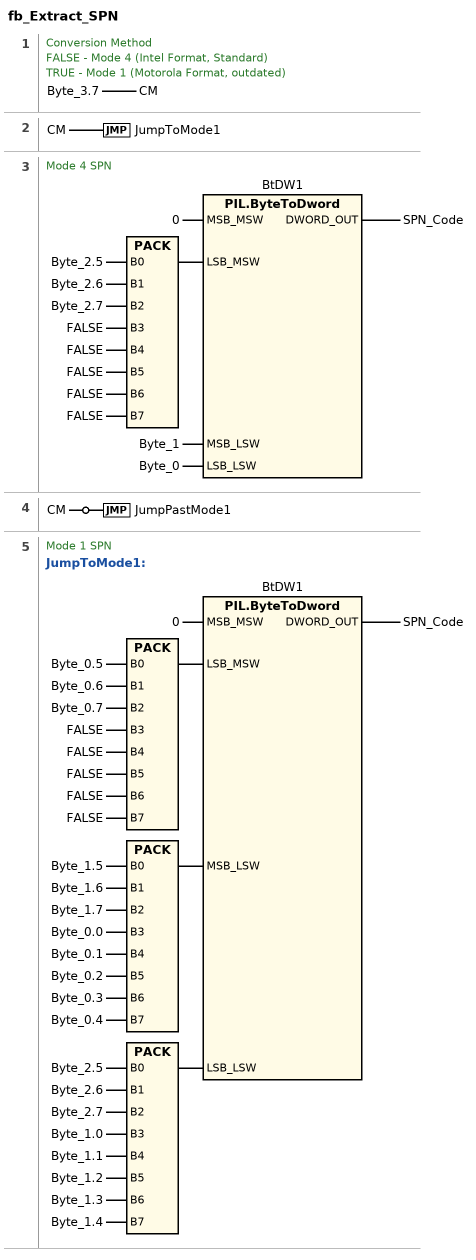
// NETWORK 1
// 					Conversion Method
// FALSE - Mode 4 (Intel Format, Standard)
// TRUE - Mode 1 (Motorola Format, outdated)
//
CM := Byte_3.7;

// NETWORK 2
IF CM THEN JMP JumpToMode1; END_IF

// NETWORK 3
// Mode 4 SPN
BtDW1(
    MSB_MSW := 0,
    LSB_MSW := PACK(B0 := Byte_2.5, B1 := Byte_2.6, B2 := Byte_2.7, B3 := FALSE, B4 := FALSE, B5 := FALSE, B6 := FALSE, B7 := FALSE),
    MSB_LSW := Byte_1,
    LSB_LSW := Byte_0); // PIL.ByteToDword
SPN_Code := BtDW1.DWORD_OUT;

// NETWORK 4
IF NOT CM THEN JMP JumpPastMode1; END_IF

// NETWORK 5
// Mode 1 SPN
JumpToMode1:
BtDW1(
    MSB_MSW := 0,
    LSB_MSW := PACK(B0 := Byte_0.5, B1 := Byte_0.6, B2 := Byte_0.7, B3 := FALSE, B4 := FALSE, B5 := FALSE, B6 := FALSE, B7 := FALSE),
    MSB_LSW := PACK(B0 := Byte_1.5, B1 := Byte_1.6, B2 := Byte_1.7, B3 := Byte_0.0, B4 := Byte_0.1, B5 := Byte_0.2, B6 := Byte_0.3, B7 := Byte_0.4),
    LSB_LSW := PACK(B0 := Byte_2.5, B1 := Byte_2.6, B2 := Byte_2.7, B3 := Byte_1.0, B4 := Byte_1.1, B5 := Byte_1.2, B6 := Byte_1.3, B7 := Byte_1.4)); // PIL.ByteToDword
SPN_Code := BtDW1.DWORD_OUT;

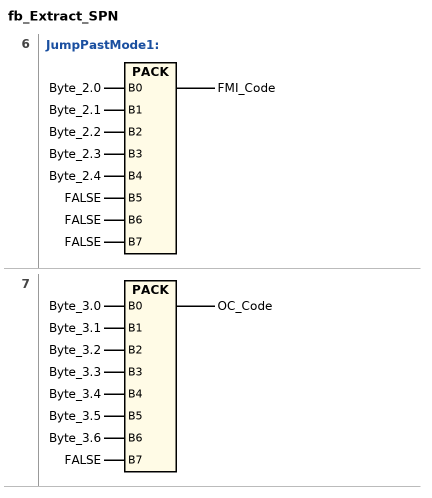
// NETWORK 6
JumpPastMode1:
FMI_Code := PACK(B0 := Byte_2.0, B1 := Byte_2.1, B2 := Byte_2.2, B3 := Byte_2.3, B4 := Byte_2.4, B5 := FALSE, B6 := FALSE, B7 := FALSE);

// NETWORK 7
OC_Code := PACK(B0 := Byte_3.0, B1 := Byte_3.1, B2 := Byte_3.2, B3 := Byte_3.3, B4 := Byte_3.4, B5 := Byte_3.5, B6 := Byte_3.6, B7 := FALSE);

END_FUNCTION_BLOCK

// Device/Application/App_PLC/CAN Comms/Engine Comms/Pack2bits
FUNCTION_BLOCK Pack2bits
VAR_INPUT
	LS_bit: BOOL;
	MS_bit: BOOL;
END_VAR
VAR_OUTPUT
	Out: BYTE;
END_VAR
VAR
END_VAR

IF LS_bit=TRUE THEN Out:=1; ELSE Out:=0; END_IF
IF MS_bit=TRUE THEN Out:=Out+2; ELSE Out:=Out; END_IF

END_FUNCTION_BLOCK

// Device/Application/App_PLC/CAN Comms/Engine Comms/PLC_DM1_Condition
FUNCTION_BLOCK PLC_DM1_Condition

(*Function block to look for an active SPN that is contained within the Error codes array [1..15]
The ConditionActive ouptut is used when you want to identify a SPN with a certain FMI
The SPNActive output is TRUE when the requested SPN is contained anywhere withing the array*)

VAR_INPUT
	ActiveErrCount: BYTE;
	ReqSPN: DWORD;
	ReqFMI: BYTE;
END_VAR
VAR_OUTPUT
	SPNActive: BOOL;
	ConditionAcitve: BOOL;
END_VAR
VAR
(*Temporary Variables*)
	SPNActive_1: BOOL;
	SPNActive_2: BOOL;
	SPNActive_3: BOOL;
	SPNActive_4: BOOL;
	SPNActive_5: BOOL;
	SPNActive_6: BOOL;
	SPNActive_7: BOOL;	(*  *)
	SPNActive_8: BOOL;	(*  *)
END_VAR
VAR // added by the converter: edge detectors and wires of the graphical bodies
    _w1, _w2, _w3, _w4, _w5, _w6, _w7, _w8 : BOOL;
END_VAR

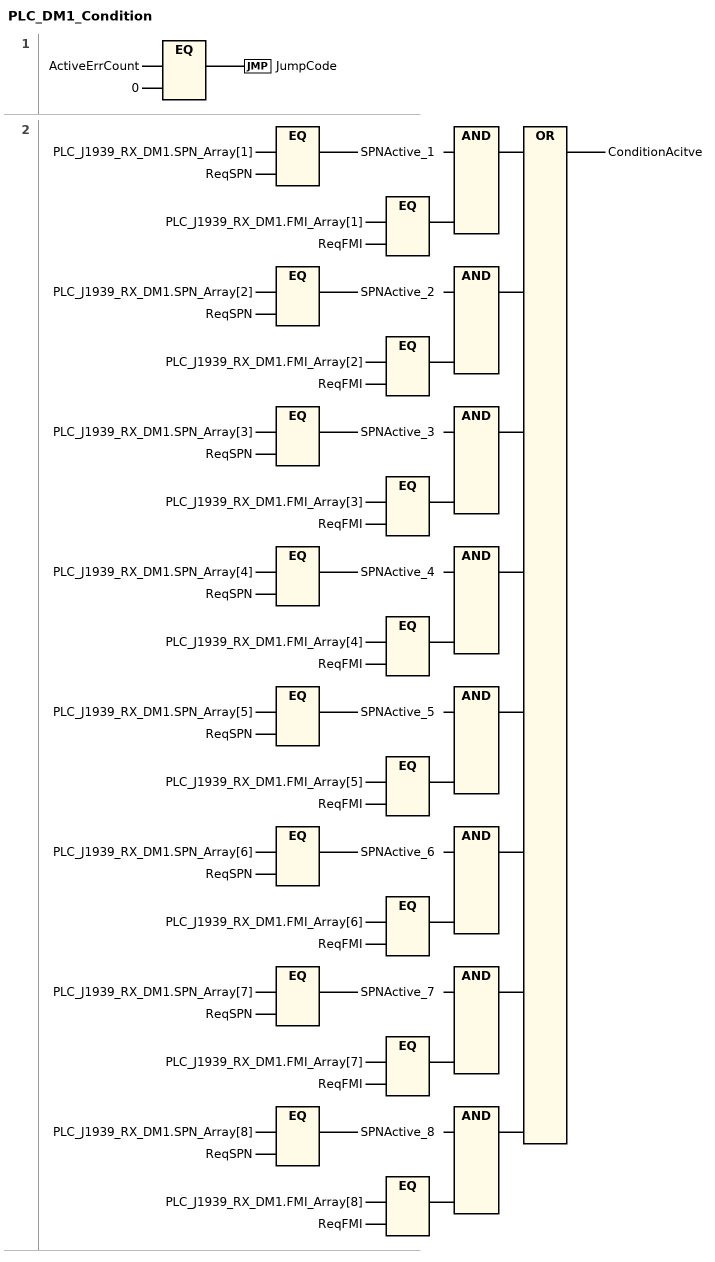
// NETWORK 1
IF ActiveErrCount = 0 THEN JMP JumpCode; END_IF

// NETWORK 2
_w1 := PLC_J1939_RX_DM1.SPN_Array[1] = ReqSPN;
SPNActive_1 := _w1;
_w2 := PLC_J1939_RX_DM1.SPN_Array[2] = ReqSPN;
SPNActive_2 := _w2;
_w3 := PLC_J1939_RX_DM1.SPN_Array[3] = ReqSPN;
SPNActive_3 := _w3;
_w4 := PLC_J1939_RX_DM1.SPN_Array[4] = ReqSPN;
SPNActive_4 := _w4;
_w5 := PLC_J1939_RX_DM1.SPN_Array[5] = ReqSPN;
SPNActive_5 := _w5;
_w6 := PLC_J1939_RX_DM1.SPN_Array[6] = ReqSPN;
SPNActive_6 := _w6;
_w7 := PLC_J1939_RX_DM1.SPN_Array[7] = ReqSPN;
SPNActive_7 := _w7;
_w8 := PLC_J1939_RX_DM1.SPN_Array[8] = ReqSPN;
SPNActive_8 := _w8;
ConditionAcitve := _w1 AND PLC_J1939_RX_DM1.FMI_Array[1] = ReqFMI OR _w2 AND PLC_J1939_RX_DM1.FMI_Array[2] = ReqFMI OR _w3 AND PLC_J1939_RX_DM1.FMI_Array[3] = ReqFMI OR _w4 AND PLC_J1939_RX_DM1.FMI_Array[4] = ReqFMI OR _w5 AND PLC_J1939_RX_DM1.FMI_Array[5] = ReqFMI OR _w6 AND PLC_J1939_RX_DM1.FMI_Array[6] = ReqFMI OR _w7 AND PLC_J1939_RX_DM1.FMI_Array[7] = ReqFMI OR _w8 AND PLC_J1939_RX_DM1.FMI_Array[8] = ReqFMI;

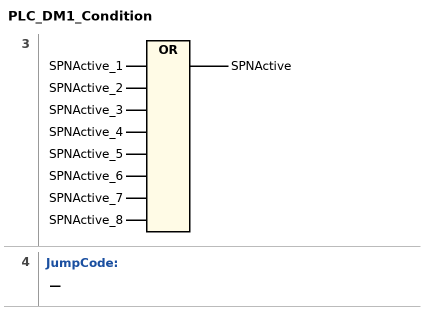
// NETWORK 3
SPNActive := SPNActive_1 OR SPNActive_2 OR SPNActive_3 OR SPNActive_4 OR SPNActive_5 OR SPNActive_6 OR SPNActive_7 OR SPNActive_8;

// NETWORK 4
JumpCode: ;

END_FUNCTION_BLOCK

// Device/Application/App_Common/Machine/APP_WARNINGS_ERRORS
PROGRAM APP_WARNINGS_ERRORS
VAR_INPUT
	TOTAL_ERRORS:INT;
	TOTAL_WARNINGS:INT;	
END_VAR
VAR
	HEADER_MSG_SWT_TON: TON;
	HEADER_MSG_SWT: WORD;
	HEADER_MSG_ENA: BOOL:=TRUE;

END_VAR
VAR_OUTPUT
	ERRORS_ACTIVE: BOOL;
	WARNINGS_ACTIVE: BOOL;
END_VAR


//TOTAL_ERRORS:=MAIN_ERRORS_COUNT+DIAG_IO_ERRORS_COUNT;

IF TOTAL_ERRORS > 0 THEN
	ERRORS_ACTIVE:=TRUE;
ELSE
	ERRORS_ACTIVE:=FALSE;
END_IF

IF TOTAL_WARNINGS > 0 THEN
	WARNINGS_ACTIVE:=TRUE;
ELSE
	WARNINGS_ACTIVE:=FALSE;
END_IF

IF HEADER_MSG_ENA THEN
	HEADER_MSG_SWT_TON(IN:=NOT(HEADER_MSG_SWT_TON.Q));
	
	IF HEADER_MSG_SWT_TON.Q THEN
		IF HEADER_MSG_SWT < 2 THEN
			HEADER_MSG_SWT:=HEADER_MSG_SWT+1;	
		ELSE
			HEADER_MSG_SWT:=0;		
		END_IF	
	END_IF

	IF GVL_Alarms.EMERGENCY_STOP_COMMON AND HEADER_MSG_SWT = 1 THEN
		NVL_Viz.Sections.Footer.Header_Message_Str:='ESTOP ACTIVE';
		NVL_Viz.Sections.Footer.Header_Message_Colour:=16#FFFF0000;
		NVL_Viz.Sections.Footer.Header_Message_Show:=TRUE;
		HEADER_MSG_SWT_TON.PT:=T#2000MS;
	ELSIF GVL_Alarms.ETHERNET_PLC_COMMON_FAILURE AND HEADER_MSG_SWT = 2 THEN
		NVL_Viz.Sections.Footer.Header_Message_Str:='PLCS OFFLINE';
		NVL_Viz.Sections.Footer.Header_Message_Colour:=16#FFFF0000;
		NVL_Viz.Sections.Footer.Header_Message_Show:=TRUE;
		HEADER_MSG_SWT_TON.PT:=T#3000MS;
	ELSE
		NVL_Viz.Sections.Footer.Header_Message_Str:='';
		NVL_Viz.Sections.Footer.Header_Message_Colour:=16#FF000000;
		NVL_Viz.Sections.Footer.Header_Message_Show:=FALSE;	
		HEADER_MSG_SWT_TON.PT:=T#1000MS;
	END_IF
ELSE
	NVL_Viz.Sections.Footer.Header_Message_Show:=FALSE;	
END_IF

END_PROGRAM

// Device/Application/App_Common/Machine/SIREN_BEACONS
PROGRAM SIREN_BEACONS
VAR_INPUT
	ESTOP_ACTIVE: BOOL;
	ERRORS_ACTIVE: BOOL;
	WARNINGS_ACTIVE: BOOL;
END_VAR
VAR
	SIREN_BLIP_PU_TON: TON;
	PRE_START_TON: TON;	
	
	SIREN_ALARMS: BOOL:=FALSE;
	SIREN_WARNINGS: BOOL:=FALSE;

	SIREN_PU_BLIP: BOOL;
	BEACON_PU_BLIP: BOOL;	
	
	BEACON_DEADMAN: BOOL;
	SIREN_DEADMAN: BOOL;
	SIREN_ESTOP: BOOL;
	TEST_SIREN: BOOL;
	TEST_BEACON: BOOL;
	
	SIREN_ALARMS_BLINK: DUTY_CYCLE;
	SIREN_WARNINGS_BLINK: DUTY_CYCLE;
END_VAR

VAR_OUTPUT
	SIREN_OUT: BOOL;
	BEACON_OUT: BOOL;
	PRESTART_TIMER_ACTIVE: BOOL;	
	PRESTART_TIMER_DONE: BOOL;
END_VAR
VAR // added by the converter: edge detectors and wires of the graphical bodies
    _w1 : BOOL;
END_VAR

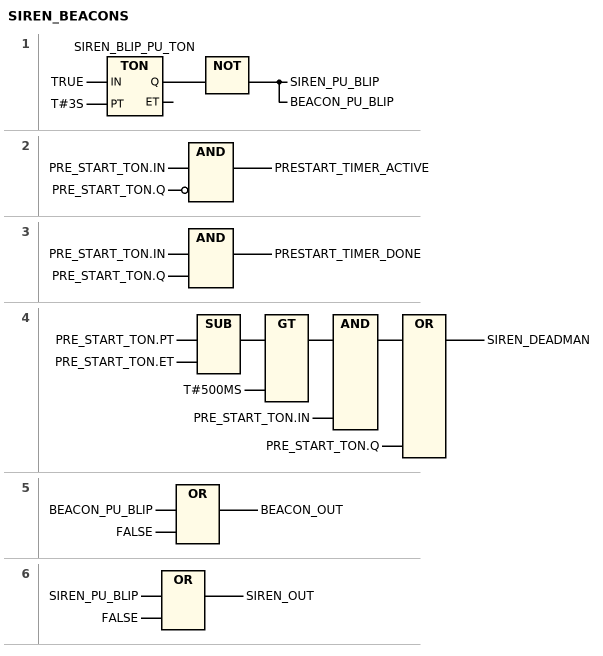
// NETWORK 1
SIREN_BLIP_PU_TON(IN := TRUE, PT := T#3S); // TON
_w1 := NOT SIREN_BLIP_PU_TON.Q;
SIREN_PU_BLIP := _w1;
BEACON_PU_BLIP := _w1;

// NETWORK 2
PRESTART_TIMER_ACTIVE := PRE_START_TON.IN AND NOT PRE_START_TON.Q;

// NETWORK 3
PRESTART_TIMER_DONE := PRE_START_TON.IN AND PRE_START_TON.Q;

// NETWORK 4
SIREN_DEADMAN := PRE_START_TON.PT - PRE_START_TON.ET > T#500MS AND PRE_START_TON.IN OR PRE_START_TON.Q;

// NETWORK 5
BEACON_OUT := BEACON_PU_BLIP OR FALSE;

// NETWORK 6
SIREN_OUT := SIREN_PU_BLIP OR FALSE;

END_PROGRAM

// Device/Application/App_Common/Nav/Page Control/AutoManSelButtons
PROGRAM AutoManSelButtons
VAR_INPUT
	Enable: BOOL;	
END_VAR

VAR
	Mimic_Halo_Sel_Max: WORD:=6;
	NavUpShow_TP: TP;
	NavDownShow_TP: TP;
	NavCircleShow_TP: TP;
	TailConv_RectIcon_FB: RectIcon;
	SideTransfer_RectIcon_FB: RectIcon;
	SideConveyor_RectIcon_FB: RectIcon;
	CollectConveyor_RectIcon_FB: RectIcon;
	Drum_RectIcon_FB: RectIcon;
	Feeder_RectIcon_FB: RectIcon;
	NavLeftShow_TP: TP;
	NavRightShow_TP: TP;
	AUTOSTOP_DUTY_CYCLE: DUTY_CYCLE;
	AUTOSTART_DUTY_CYCLE: DUTY_CYCLE;
	AutoActiveCommon: BOOL;
	
	PWM_Op_Status_FB_0: PWM_Op_Status_FB;
	PWM_Op_Status_FB_1: PWM_Op_Status_FB;
	PWM_Op_Status_FB_2: PWM_Op_Status_FB;
	PWM_Op_Status_FB_3: PWM_Op_Status_FB;
	PWM_Op_Status_FB_4: PWM_Op_Status_FB;
	PWM_Op_Status_FB_5: PWM_Op_Status_FB;	
	PWM_Op_Status_FB_: PWM_Op_Status_FB;
	
	PWM_Op_SideConveyor_Status_Str: STRING;
	PWM_Op_SideTransfer_Status_Str: STRING;	
	PWM_Op_TailConveyor_Status_Str: STRING;
	PWM_Op_CollectionConveyor_Status_Str: STRING;
	PWM_Op_DrumSpeed_Status_Str: STRING;
	PWM_Op_FeederSpeed_Status_Str: STRING;
END_VAR

VAR_OUTPUT
	AutoStartShow: BOOL;
	AutoStopShow: BOOL;	
	Selected_String: STRING;
	NavUpShow: BOOL;
	NavDownShow: BOOL;	
	NavLeftShow: BOOL;
	NavRightShow: BOOL;	
	NavCirleShow: BOOL;	
	NavIdleShow: BOOL;
	NavSelectShow: BOOL;
	Mimic_Halo_Sel: WORD;
	Mimic_Halo_1: BOOL;
	Mimic_Halo_2: BOOL;
	Mimic_Halo_3: BOOL;
	Mimic_Halo_4: BOOL;
	Mimic_Halo_5: BOOL;
	Mimic_Halo_6: BOOL;
	Mimic_Halo_RPM_Up_Down: BOOL;	
	Button_1: BOOL;
	Button_2: BOOL;
	Button_3: BOOL;
	Button_4: BOOL;
	Button_5: BOOL;
	Button_6: BOOL;
	Button_Rpm_Up: BOOL;
	Button_Rpm_Down: BOOL;
	
	Icon_1_Fill_Colour: DWORD;
	Icon_2_Fill_Colour: DWORD;
	Icon_3_Fill_Colour: DWORD;
	Icon_4_Fill_Colour: DWORD;
	Icon_5_Fill_Colour: DWORD;
	Icon_6_Fill_Colour: DWORD;	
END_VAR
VAR // added by the converter: edge detectors and wires of the graphical bodies
    _rt1, _rt2 : R_TRIG;
    _w1, _w2, _w3, _w4, _w5, _w6, _w7 : BOOL;
END_VAR

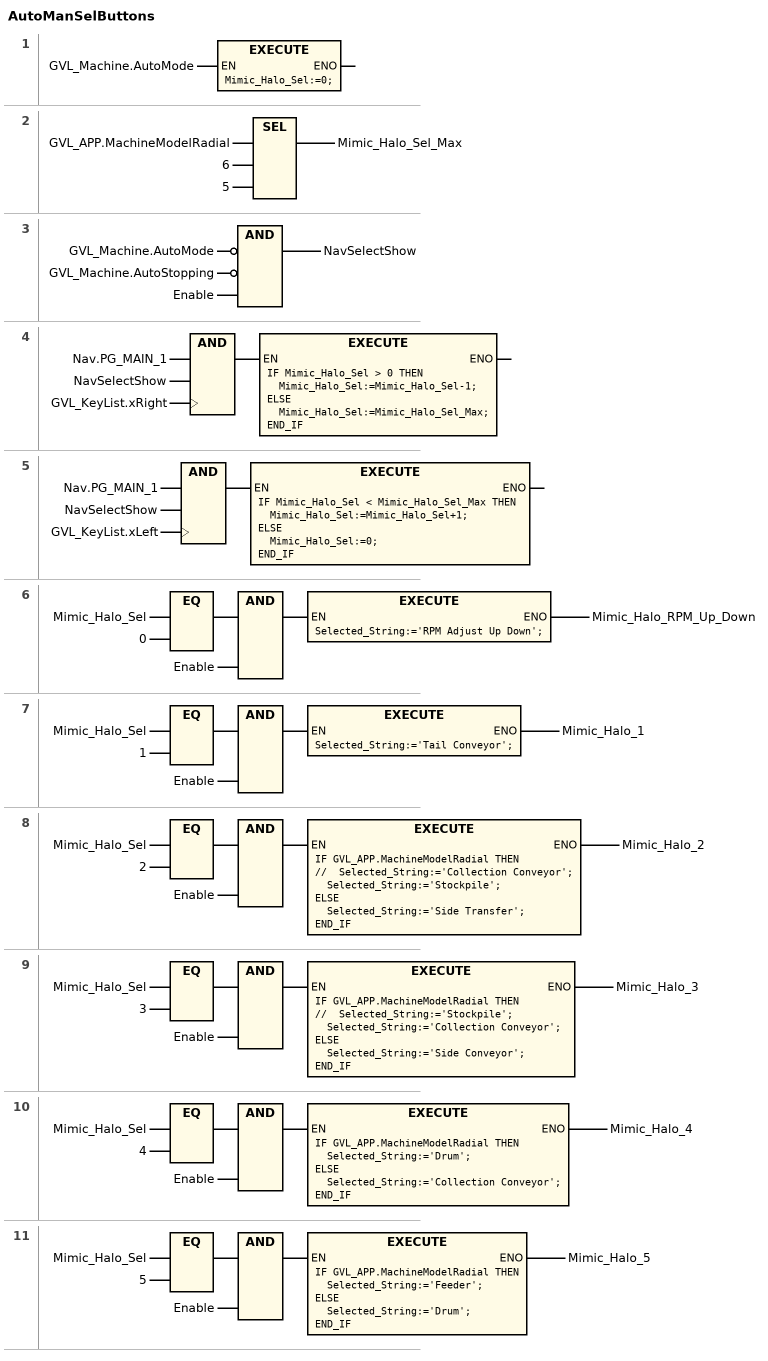
// NETWORK 1
IF GVL_Machine.AutoMode THEN Mimic_Halo_Sel:=0; END_IF

// NETWORK 2
Mimic_Halo_Sel_Max := SEL(GVL_APP.MachineModelRadial, 6, 5);

// NETWORK 3
NavSelectShow := NOT GVL_Machine.AutoMode AND NOT GVL_Machine.AutoStopping AND Enable;

// NETWORK 4
_rt1(CLK := GVL_KeyList.xRight);
IF Nav.PG_MAIN_1 AND NavSelectShow AND _rt1.Q THEN
    IF Mimic_Halo_Sel > 0 THEN 
    	Mimic_Halo_Sel:=Mimic_Halo_Sel-1;
    ELSE
    	Mimic_Halo_Sel:=Mimic_Halo_Sel_Max;
    END_IF
END_IF

// NETWORK 5
_rt2(CLK := GVL_KeyList.xLeft);
IF Nav.PG_MAIN_1 AND NavSelectShow AND _rt2.Q THEN
    IF Mimic_Halo_Sel < Mimic_Halo_Sel_Max THEN 
    	Mimic_Halo_Sel:=Mimic_Halo_Sel+1;
    ELSE
    	Mimic_Halo_Sel:=0;
    END_IF
END_IF

// NETWORK 6
_w1 := Mimic_Halo_Sel = 0 AND Enable;
IF _w1 THEN Selected_String:='RPM Adjust Up Down'; END_IF
Mimic_Halo_RPM_Up_Down := _w1;

// NETWORK 7
_w2 := Mimic_Halo_Sel = 1 AND Enable;
IF _w2 THEN Selected_String:='Tail Conveyor'; END_IF
Mimic_Halo_1 := _w2;

// NETWORK 8
_w3 := Mimic_Halo_Sel = 2 AND Enable;
IF _w3 THEN
    IF GVL_APP.MachineModelRadial THEN
    //	Selected_String:='Collection Conveyor';
    	Selected_String:='Stockpile';	
    ELSE
    	Selected_String:='Side Transfer';	
    END_IF
END_IF
Mimic_Halo_2 := _w3;

// NETWORK 9
_w4 := Mimic_Halo_Sel = 3 AND Enable;
IF _w4 THEN
    IF GVL_APP.MachineModelRadial THEN
    //	Selected_String:='Stockpile';	
    	Selected_String:='Collection Conveyor';	
    ELSE
    	Selected_String:='Side Conveyor';	
    END_IF
END_IF
Mimic_Halo_3 := _w4;

// NETWORK 10
_w5 := Mimic_Halo_Sel = 4 AND Enable;
IF _w5 THEN
    IF GVL_APP.MachineModelRadial THEN
    	Selected_String:='Drum';
    ELSE
    	Selected_String:='Collection Conveyor';
    END_IF
END_IF
Mimic_Halo_4 := _w5;

// NETWORK 11
_w6 := Mimic_Halo_Sel = 5 AND Enable;
IF _w6 THEN
    IF GVL_APP.MachineModelRadial THEN
    	Selected_String:='Feeder';
    ELSE
    	Selected_String:='Drum';		
    END_IF
END_IF
Mimic_Halo_5 := _w6;

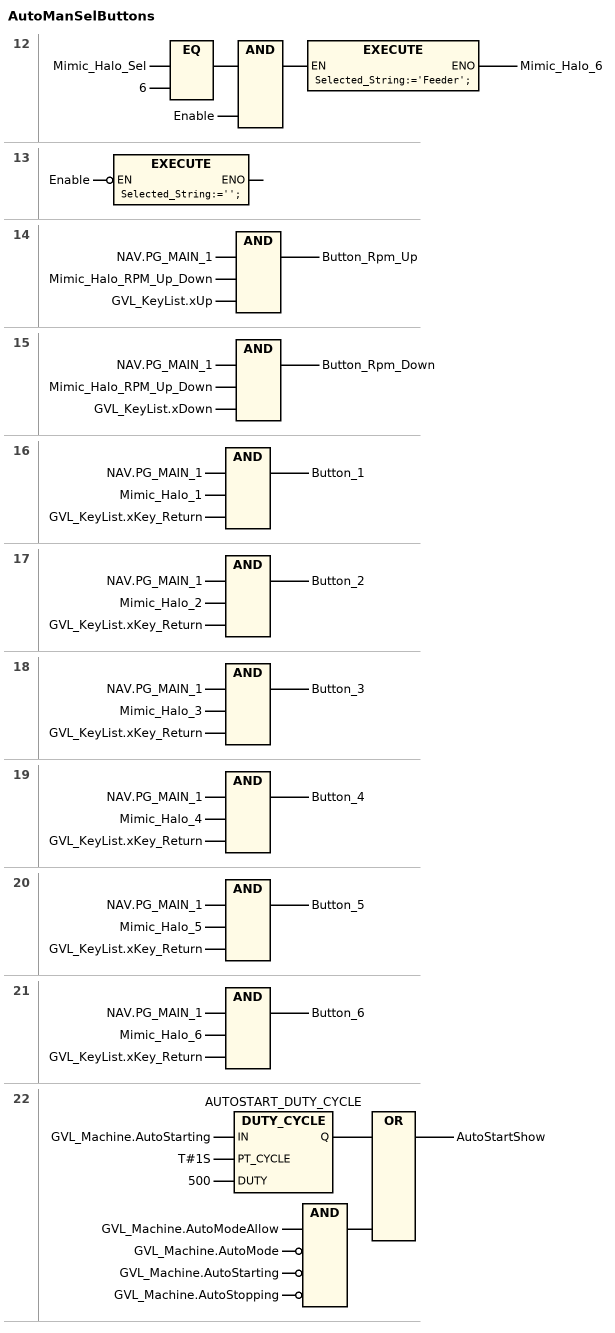
// NETWORK 12
_w7 := Mimic_Halo_Sel = 6 AND Enable;
IF _w7 THEN Selected_String:='Feeder'; END_IF
Mimic_Halo_6 := _w7;

// NETWORK 13
IF NOT Enable THEN Selected_String:=''; END_IF

// NETWORK 14
Button_Rpm_Up := NAV.PG_MAIN_1 AND Mimic_Halo_RPM_Up_Down AND GVL_KeyList.xUp;

// NETWORK 15
Button_Rpm_Down := NAV.PG_MAIN_1 AND Mimic_Halo_RPM_Up_Down AND GVL_KeyList.xDown;

// NETWORK 16
Button_1 := NAV.PG_MAIN_1 AND Mimic_Halo_1 AND GVL_KeyList.xKey_Return;

// NETWORK 17
Button_2 := NAV.PG_MAIN_1 AND Mimic_Halo_2 AND GVL_KeyList.xKey_Return;

// NETWORK 18
Button_3 := NAV.PG_MAIN_1 AND Mimic_Halo_3 AND GVL_KeyList.xKey_Return;

// NETWORK 19
Button_4 := NAV.PG_MAIN_1 AND Mimic_Halo_4 AND GVL_KeyList.xKey_Return;

// NETWORK 20
Button_5 := NAV.PG_MAIN_1 AND Mimic_Halo_5 AND GVL_KeyList.xKey_Return;

// NETWORK 21
Button_6 := NAV.PG_MAIN_1 AND Mimic_Halo_6 AND GVL_KeyList.xKey_Return;

// NETWORK 22
AUTOSTART_DUTY_CYCLE(IN := GVL_Machine.AutoStarting, PT_CYCLE := T#1S, DUTY := 500); // DUTY_CYCLE
AutoStartShow := AUTOSTART_DUTY_CYCLE.Q OR GVL_Machine.AutoModeAllow AND NOT GVL_Machine.AutoMode AND NOT GVL_Machine.AutoStarting AND NOT GVL_Machine.AutoStopping;

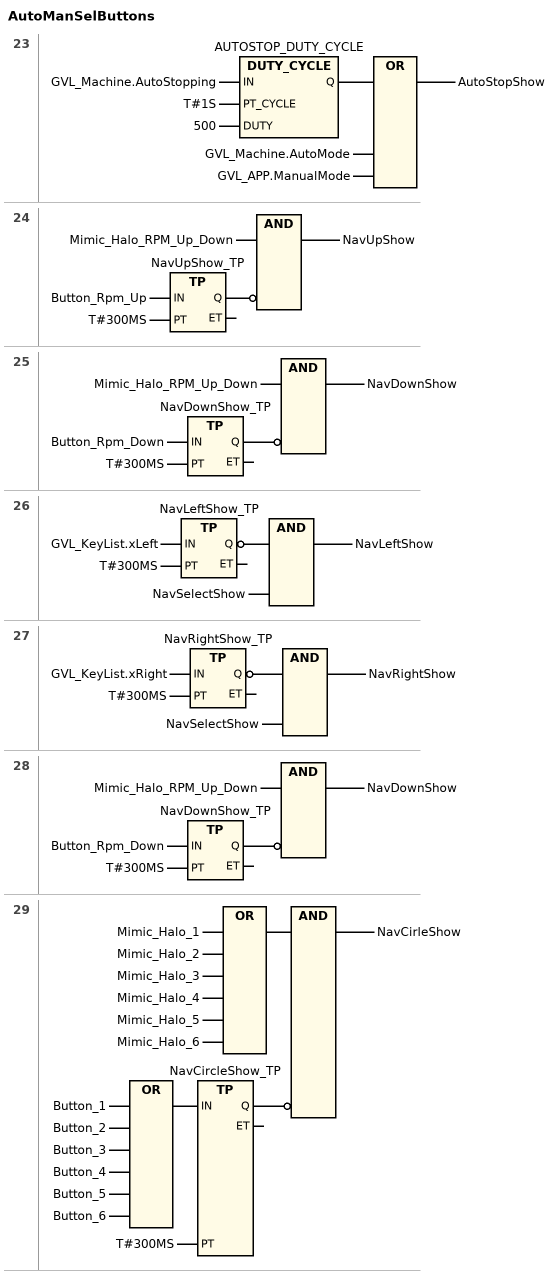
// NETWORK 23
AUTOSTOP_DUTY_CYCLE(IN := GVL_Machine.AutoStopping, PT_CYCLE := T#1S, DUTY := 500); // DUTY_CYCLE
AutoStopShow := AUTOSTOP_DUTY_CYCLE.Q OR GVL_Machine.AutoMode OR GVL_APP.ManualMode;

// NETWORK 24
NavUpShow_TP(IN := Button_Rpm_Up, PT := T#300MS); // TP
NavUpShow := Mimic_Halo_RPM_Up_Down AND NOT NavUpShow_TP.Q;

// NETWORK 25
NavDownShow_TP(IN := Button_Rpm_Down, PT := T#300MS); // TP
NavDownShow := Mimic_Halo_RPM_Up_Down AND NOT NavDownShow_TP.Q;

// NETWORK 26
NavLeftShow_TP(IN := GVL_KeyList.xLeft, PT := T#300MS); // TP
NavLeftShow := NOT NavLeftShow_TP.Q AND NavSelectShow;

// NETWORK 27
NavRightShow_TP(IN := GVL_KeyList.xRight, PT := T#300MS); // TP
NavRightShow := NOT NavRightShow_TP.Q AND NavSelectShow;

// NETWORK 28
NavDownShow_TP(IN := Button_Rpm_Down, PT := T#300MS); // TP
NavDownShow := Mimic_Halo_RPM_Up_Down AND NOT NavDownShow_TP.Q;

// NETWORK 29
NavCircleShow_TP(IN := Button_1 OR Button_2 OR Button_3 OR Button_4 OR Button_5 OR Button_6, PT := T#300MS); // TP
NavCirleShow := (Mimic_Halo_1 OR Mimic_Halo_2 OR Mimic_Halo_3 OR Mimic_Halo_4 OR Mimic_Halo_5 OR Mimic_Halo_6) AND NOT NavCircleShow_TP.Q;

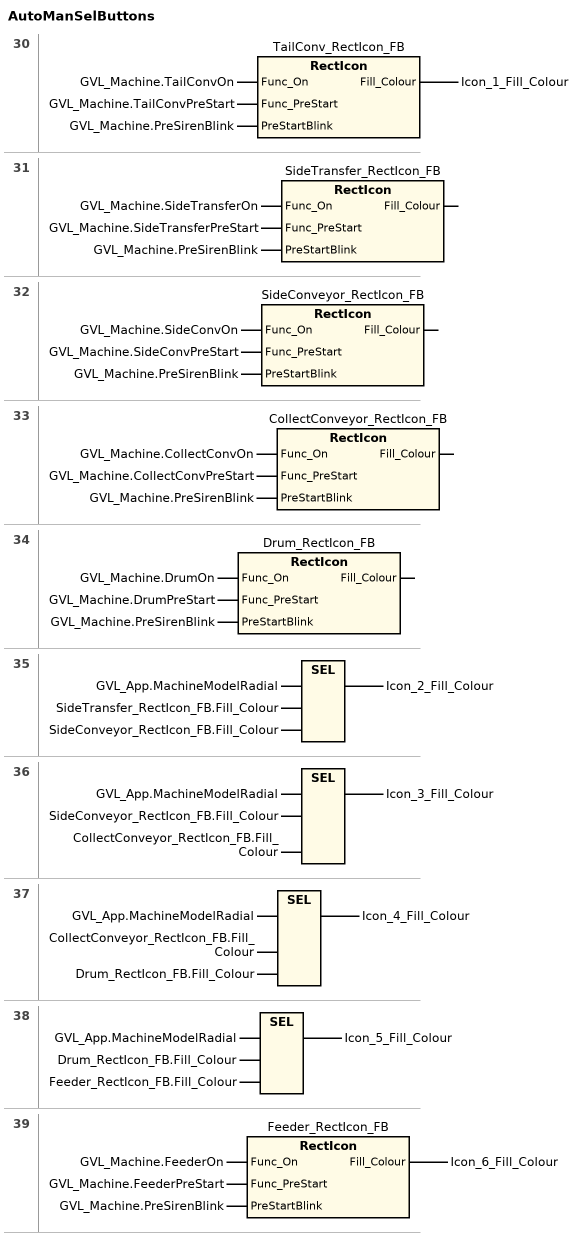
// NETWORK 30
TailConv_RectIcon_FB(
    Func_On := GVL_Machine.TailConvOn,
    Func_PreStart := GVL_Machine.TailConvPreStart,
    PreStartBlink := GVL_Machine.PreSirenBlink); // RectIcon
Icon_1_Fill_Colour := TailConv_RectIcon_FB.Fill_Colour;

// NETWORK 31
SideTransfer_RectIcon_FB(
    Func_On := GVL_Machine.SideTransferOn,
    Func_PreStart := GVL_Machine.SideTransferPreStart,
    PreStartBlink := GVL_Machine.PreSirenBlink); // RectIcon

// NETWORK 32
SideConveyor_RectIcon_FB(
    Func_On := GVL_Machine.SideConvOn,
    Func_PreStart := GVL_Machine.SideConvPreStart,
    PreStartBlink := GVL_Machine.PreSirenBlink); // RectIcon

// NETWORK 33
CollectConveyor_RectIcon_FB(
    Func_On := GVL_Machine.CollectConvOn,
    Func_PreStart := GVL_Machine.CollectConvPreStart,
    PreStartBlink := GVL_Machine.PreSirenBlink); // RectIcon

// NETWORK 34
Drum_RectIcon_FB(
    Func_On := GVL_Machine.DrumOn,
    Func_PreStart := GVL_Machine.DrumPreStart,
    PreStartBlink := GVL_Machine.PreSirenBlink); // RectIcon

// NETWORK 35
Icon_2_Fill_Colour := SEL(GVL_App.MachineModelRadial, SideTransfer_RectIcon_FB.Fill_Colour, SideConveyor_RectIcon_FB.Fill_Colour);

// NETWORK 36
Icon_3_Fill_Colour := SEL(GVL_App.MachineModelRadial, SideConveyor_RectIcon_FB.Fill_Colour, CollectConveyor_RectIcon_FB.Fill_Colour);

// NETWORK 37
Icon_4_Fill_Colour := SEL(GVL_App.MachineModelRadial, CollectConveyor_RectIcon_FB.Fill_Colour, Drum_RectIcon_FB.Fill_Colour);

// NETWORK 38
Icon_5_Fill_Colour := SEL(GVL_App.MachineModelRadial, Drum_RectIcon_FB.Fill_Colour, Feeder_RectIcon_FB.Fill_Colour);

// NETWORK 39
Feeder_RectIcon_FB(
    Func_On := GVL_Machine.FeederOn,
    Func_PreStart := GVL_Machine.FeederPreStart,
    PreStartBlink := GVL_Machine.PreSirenBlink); // RectIcon
Icon_6_Fill_Colour := Feeder_RectIcon_FB.Fill_Colour;

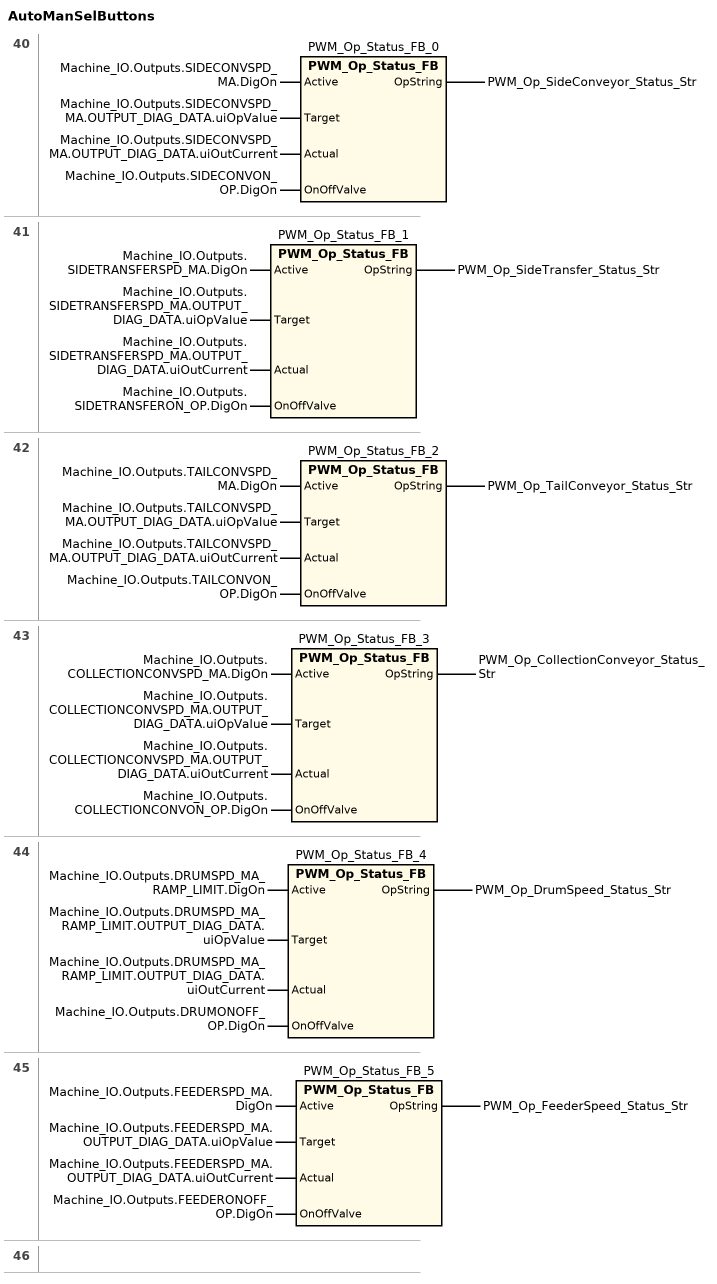
// NETWORK 40
PWM_Op_Status_FB_0(
    Active := Machine_IO.Outputs.SIDECONVSPD_MA.DigOn,
    Target := Machine_IO.Outputs.SIDECONVSPD_MA.OUTPUT_DIAG_DATA.uiOpValue,
    Actual := Machine_IO.Outputs.SIDECONVSPD_MA.OUTPUT_DIAG_DATA.uiOutCurrent,
    OnOffValve := Machine_IO.Outputs.SIDECONVON_OP.DigOn); // PWM_Op_Status_FB
PWM_Op_SideConveyor_Status_Str := PWM_Op_Status_FB_0.OpString;

// NETWORK 41
PWM_Op_Status_FB_1(
    Active := Machine_IO.Outputs.SIDETRANSFERSPD_MA.DigOn,
    Target := Machine_IO.Outputs.SIDETRANSFERSPD_MA.OUTPUT_DIAG_DATA.uiOpValue,
    Actual := Machine_IO.Outputs.SIDETRANSFERSPD_MA.OUTPUT_DIAG_DATA.uiOutCurrent,
    OnOffValve := Machine_IO.Outputs.SIDETRANSFERON_OP.DigOn); // PWM_Op_Status_FB
PWM_Op_SideTransfer_Status_Str := PWM_Op_Status_FB_1.OpString;

// NETWORK 42
PWM_Op_Status_FB_2(
    Active := Machine_IO.Outputs.TAILCONVSPD_MA.DigOn,
    Target := Machine_IO.Outputs.TAILCONVSPD_MA.OUTPUT_DIAG_DATA.uiOpValue,
    Actual := Machine_IO.Outputs.TAILCONVSPD_MA.OUTPUT_DIAG_DATA.uiOutCurrent,
    OnOffValve := Machine_IO.Outputs.TAILCONVON_OP.DigOn); // PWM_Op_Status_FB
PWM_Op_TailConveyor_Status_Str := PWM_Op_Status_FB_2.OpString;

// NETWORK 43
PWM_Op_Status_FB_3(
    Active := Machine_IO.Outputs.COLLECTIONCONVSPD_MA.DigOn,
    Target := Machine_IO.Outputs.COLLECTIONCONVSPD_MA.OUTPUT_DIAG_DATA.uiOpValue,
    Actual := Machine_IO.Outputs.COLLECTIONCONVSPD_MA.OUTPUT_DIAG_DATA.uiOutCurrent,
    OnOffValve := Machine_IO.Outputs.COLLECTIONCONVON_OP.DigOn); // PWM_Op_Status_FB
PWM_Op_CollectionConveyor_Status_Str := PWM_Op_Status_FB_3.OpString;

// NETWORK 44
PWM_Op_Status_FB_4(
    Active := Machine_IO.Outputs.DRUMSPD_MA_RAMP_LIMIT.DigOn,
    Target := Machine_IO.Outputs.DRUMSPD_MA_RAMP_LIMIT.OUTPUT_DIAG_DATA.uiOpValue,
    Actual := Machine_IO.Outputs.DRUMSPD_MA_RAMP_LIMIT.OUTPUT_DIAG_DATA.uiOutCurrent,
    OnOffValve := Machine_IO.Outputs.DRUMONOFF_OP.DigOn); // PWM_Op_Status_FB
PWM_Op_DrumSpeed_Status_Str := PWM_Op_Status_FB_4.OpString;

// NETWORK 45
PWM_Op_Status_FB_5(
    Active := Machine_IO.Outputs.FEEDERSPD_MA.DigOn,
    Target := Machine_IO.Outputs.FEEDERSPD_MA.OUTPUT_DIAG_DATA.uiOpValue,
    Actual := Machine_IO.Outputs.FEEDERSPD_MA.OUTPUT_DIAG_DATA.uiOutCurrent,
    OnOffValve := Machine_IO.Outputs.FEEDERONOFF_OP.DigOn); // PWM_Op_Status_FB
PWM_Op_FeederSpeed_Status_Str := PWM_Op_Status_FB_5.OpString;

// NETWORK 46

END_PROGRAM

// Device/Application/App_Common/Nav/Page Control/RectIcon
FUNCTION_BLOCK RectIcon
VAR_INPUT
	Func_On: BOOL;
	Func_PreStart: BOOL;
	PreStartBlink: BOOL;
END_VAR
VAR_OUTPUT
	Fill_Colour: DWORD;
END_VAR
VAR
END_VAR

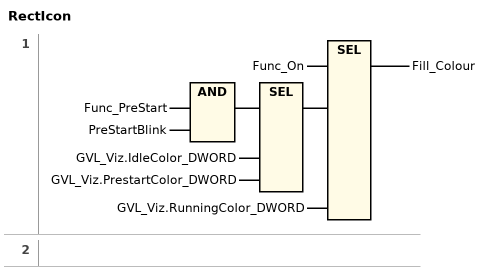
// NETWORK 1
Fill_Colour := SEL(Func_On, SEL(Func_PreStart AND PreStartBlink, GVL_Viz.IdleColor_DWORD, GVL_Viz.PrestartColor_DWORD), GVL_Viz.RunningColor_DWORD);

// NETWORK 2

END_FUNCTION_BLOCK

// Device/Application/App_Common/Nav/Page Control/PWM_Op_Status_FB
FUNCTION_BLOCK PWM_Op_Status_FB
VAR_INPUT
	Active: BOOL;
	Target: REAL;
	Actual: REAL;
	OnOffValve:BOOL;
END_VAR

VAR
	FormatString1: STRING:=' Trg.%.0fmA,';
	FormatString2: STRING:='Act.%.0fmA';
	TempString1: STRING;
	TempString2: STRING;	
	Sprintf_Result1: INT;
	Sprintf_Result2: INT;
END_VAR

VAR_OUTPUT
	OpString: STRING;
END_VAR

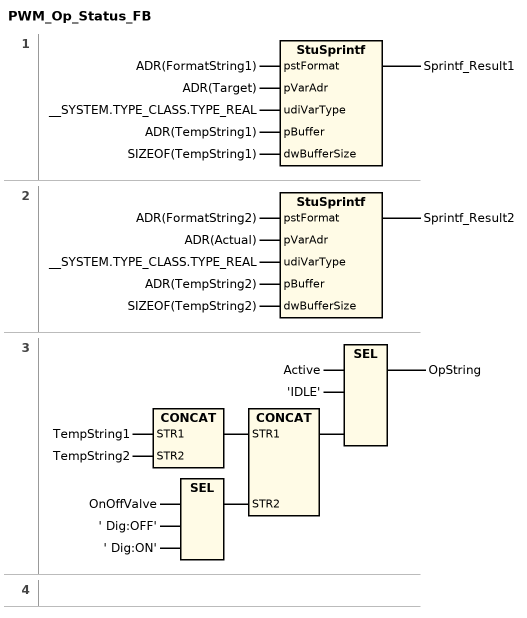
// NETWORK 1
Sprintf_Result1 := StuSprintf(pstFormat := ADR(FormatString1), pVarAdr := ADR(Target), udiVarType := __SYSTEM.TYPE_CLASS.TYPE_REAL, pBuffer := ADR(TempString1), dwBufferSize := SIZEOF(TempString1));

// NETWORK 2
Sprintf_Result2 := StuSprintf(pstFormat := ADR(FormatString2), pVarAdr := ADR(Actual), udiVarType := __SYSTEM.TYPE_CLASS.TYPE_REAL, pBuffer := ADR(TempString2), dwBufferSize := SIZEOF(TempString2));

// NETWORK 3
OpString := SEL(Active, 'IDLE', CONCAT(STR1 := CONCAT(STR1 := TempString1, STR2 := TempString2), STR2 := SEL(OnOffValve, ' Dig:OFF', ' Dig:ON')));

// NETWORK 4

END_FUNCTION_BLOCK

// Device/Application/App_PLC/Control/PLC_ManualSequence
PROGRAM PLC_ManualSequence

VAR_INPUT
	Manual_Btn_1: BOOL;
	Manual_Btn_2: BOOL;	
	Manual_Btn_3: BOOL;
	Manual_Btn_4: BOOL;
	Manual_Btn_5: BOOL;
	Manual_Btn_6: BOOL;
END_VAR

VAR
	PreSiren: BOOL;
	
	TailConv_PB: pil.PB_Toggle;
	TailConv_PreStart_TON: TON;
	TailConv_ScaleCurrent: pil.ScaleBlock;	

	SideConv_PB: pil.PB_Toggle;
	SideConv_PreStart_TON: TON;
	SideConv_ScaleCurrent: pil.ScaleBlock;
	
	SideTransfer_PB: pil.PB_Toggle;
	SideTransfer_PreStart_TON: TON;
	SideTransfer_ScaleCurrent: pil.ScaleBlock;	

	CollectConv_PB: pil.PB_Toggle;
	CollectConv_PreStart_TON: TON;
	CollectConv_ScaleCurrent: pil.ScaleBlock;

	Drum_PB: pil.PB_Toggle;
	Drum_PreStart_TON: TON;
	Drum_ScaleCurrent: pil.ScaleBlock;

	RAMP_DRUM_SP_OP: UTIL.RAMP_INT;
	RAMP_DRUM_SP_OP_ASCEND: INT:=1000;
	RAMP_DRUM_SP_OP_DESCEND: INT:=100;
	RAMP_DRUM_SP_OP_TIME_BASE: TIME:=T#1S;
	RAMP_DRUM_SP_OP_TIME_RESET: BOOL;
	DRUMSPD_MA_RAW: UINT;

	Feeder_PB: pil.PB_Toggle;
	Feeder_ScaleCurrent: pil.ScaleBlock;

	HydSetup_PB: pil.PB_Toggle;

	TailConv_OP_TON: ton;
	SideConv_OP_TON: ton;
	SideTransfer_OP_TON: ton;
	CollectConv_OP_TON: ton;
	Drum_OP_TON: ton;
	Feeder_OP_TON: ton;
	Drum_OP_Raw_TOF: TOF;
	
	// mods to help with the ramp down function for the trommel - stop damage to the valves 2-12-2024
	SetupDumpValve_PreStart_TON: TON;
	Feeder_PreStart_TON: TON;
	Common_Func_RESET: BOOL;
	TailConvSpd_Write_Test: BOOL;
END_VAR
VAR // added by the converter: edge detectors and wires of the graphical bodies
    _w1, _w2 : BOOL;
    _rt1 : R_TRIG;
END_VAR

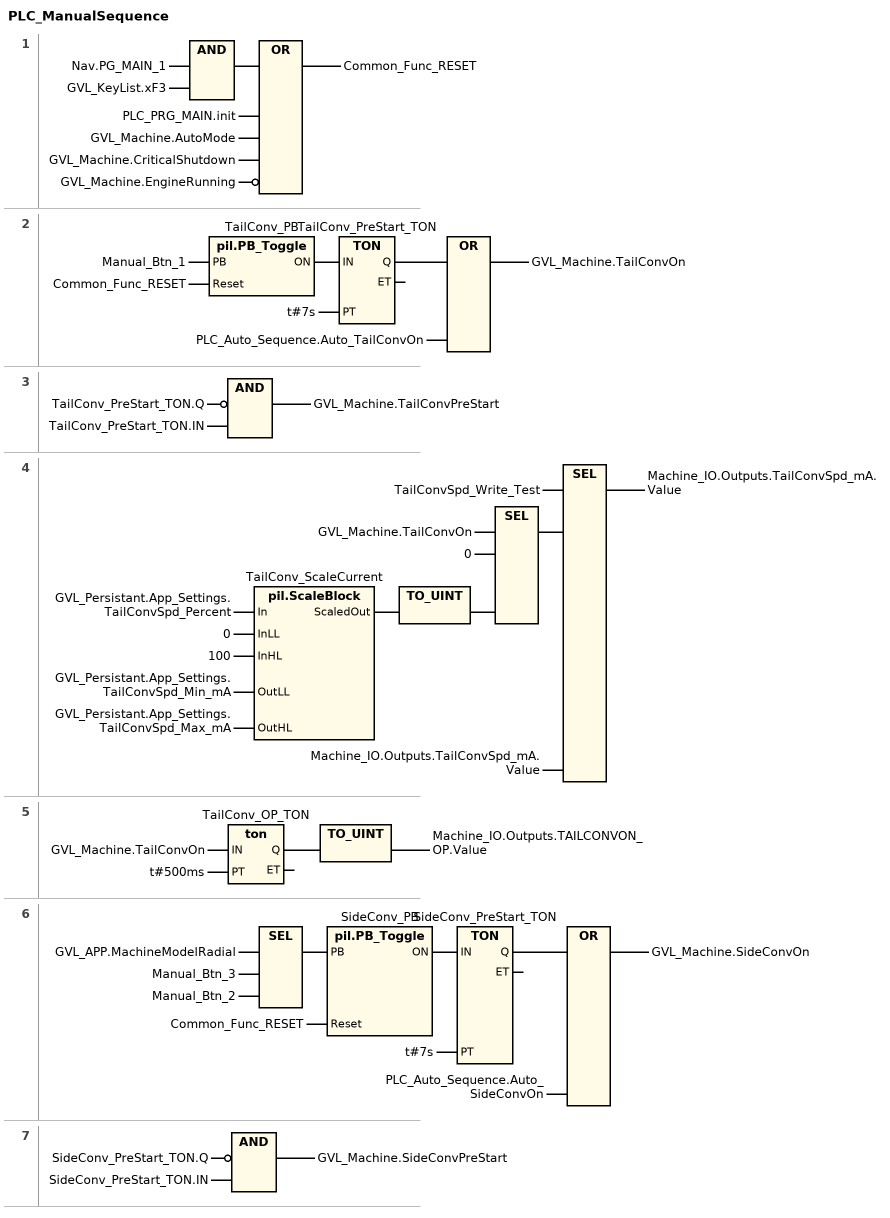
// NETWORK 1
Common_Func_RESET := Nav.PG_MAIN_1 AND GVL_KeyList.xF3 OR PLC_PRG_MAIN.init OR GVL_Machine.AutoMode OR GVL_Machine.CriticalShutdown OR NOT GVL_Machine.EngineRunning;

// NETWORK 2
TailConv_PB(PB := Manual_Btn_1, Reset := Common_Func_RESET); // pil.PB_Toggle
TailConv_PreStart_TON(IN := TailConv_PB.ON, PT := t#7s); // TON
GVL_Machine.TailConvOn := TailConv_PreStart_TON.Q OR PLC_Auto_Sequence.Auto_TailConvOn;

// NETWORK 3
GVL_Machine.TailConvPreStart := NOT TailConv_PreStart_TON.Q AND TailConv_PreStart_TON.IN;

// NETWORK 4
TailConv_ScaleCurrent(
    In := GVL_Persistant.App_Settings.TailConvSpd_Percent,
    InLL := 0,
    InHL := 100,
    OutLL := GVL_Persistant.App_Settings.TailConvSpd_Min_mA,
    OutHL := GVL_Persistant.App_Settings.TailConvSpd_Max_mA); // pil.ScaleBlock
Machine_IO.Outputs.TailConvSpd_mA.Value := SEL(TailConvSpd_Write_Test, SEL(GVL_Machine.TailConvOn, 0, TO_UINT(TailConv_ScaleCurrent.ScaledOut)), Machine_IO.Outputs.TailConvSpd_mA.Value);

// NETWORK 5
TailConv_OP_TON(IN := GVL_Machine.TailConvOn, PT := t#500ms); // ton
Machine_IO.Outputs.TAILCONVON_OP.Value := TO_UINT(TailConv_OP_TON.Q);

// NETWORK 6
SideConv_PB(PB := SEL(GVL_APP.MachineModelRadial, Manual_Btn_3, Manual_Btn_2), Reset := Common_Func_RESET); // pil.PB_Toggle
SideConv_PreStart_TON(IN := SideConv_PB.ON, PT := t#7s); // TON
GVL_Machine.SideConvOn := SideConv_PreStart_TON.Q OR PLC_Auto_Sequence.Auto_SideConvOn;

// NETWORK 7
GVL_Machine.SideConvPreStart := NOT SideConv_PreStart_TON.Q AND SideConv_PreStart_TON.IN;

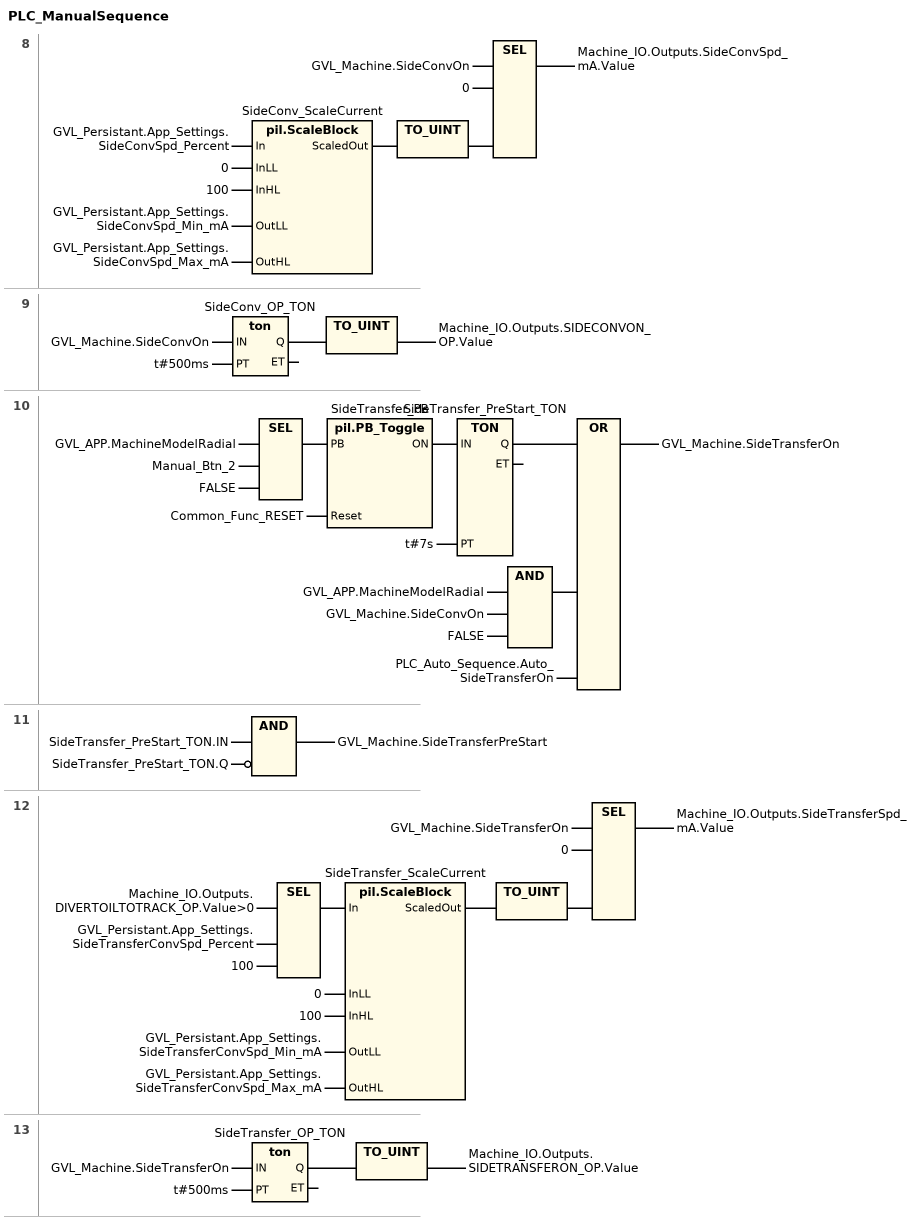
// NETWORK 8
SideConv_ScaleCurrent(
    In := GVL_Persistant.App_Settings.SideConvSpd_Percent,
    InLL := 0,
    InHL := 100,
    OutLL := GVL_Persistant.App_Settings.SideConvSpd_Min_mA,
    OutHL := GVL_Persistant.App_Settings.SideConvSpd_Max_mA); // pil.ScaleBlock
Machine_IO.Outputs.SideConvSpd_mA.Value := SEL(GVL_Machine.SideConvOn, 0, TO_UINT(SideConv_ScaleCurrent.ScaledOut));

// NETWORK 9
SideConv_OP_TON(IN := GVL_Machine.SideConvOn, PT := t#500ms); // ton
Machine_IO.Outputs.SIDECONVON_OP.Value := TO_UINT(SideConv_OP_TON.Q);

// NETWORK 10
SideTransfer_PB(PB := SEL(GVL_APP.MachineModelRadial, Manual_Btn_2, FALSE), Reset := Common_Func_RESET); // pil.PB_Toggle
SideTransfer_PreStart_TON(IN := SideTransfer_PB.ON, PT := t#7s); // TON
GVL_Machine.SideTransferOn := SideTransfer_PreStart_TON.Q OR GVL_APP.MachineModelRadial AND GVL_Machine.SideConvOn AND FALSE OR PLC_Auto_Sequence.Auto_SideTransferOn;

// NETWORK 11
GVL_Machine.SideTransferPreStart := SideTransfer_PreStart_TON.IN AND NOT SideTransfer_PreStart_TON.Q;

// NETWORK 12
SideTransfer_ScaleCurrent(
    In := SEL(Machine_IO.Outputs.DIVERTOILTOTRACK_OP.Value>0, GVL_Persistant.App_Settings.SideTransferConvSpd_Percent, 100),
    InLL := 0,
    InHL := 100,
    OutLL := GVL_Persistant.App_Settings.SideTransferConvSpd_Min_mA,
    OutHL := GVL_Persistant.App_Settings.SideTransferConvSpd_Max_mA); // pil.ScaleBlock
Machine_IO.Outputs.SideTransferSpd_mA.Value := SEL(GVL_Machine.SideTransferOn, 0, TO_UINT(SideTransfer_ScaleCurrent.ScaledOut));

// NETWORK 13
SideTransfer_OP_TON(IN := GVL_Machine.SideTransferOn, PT := t#500ms); // ton
Machine_IO.Outputs.SIDETRANSFERON_OP.Value := TO_UINT(SideTransfer_OP_TON.Q);

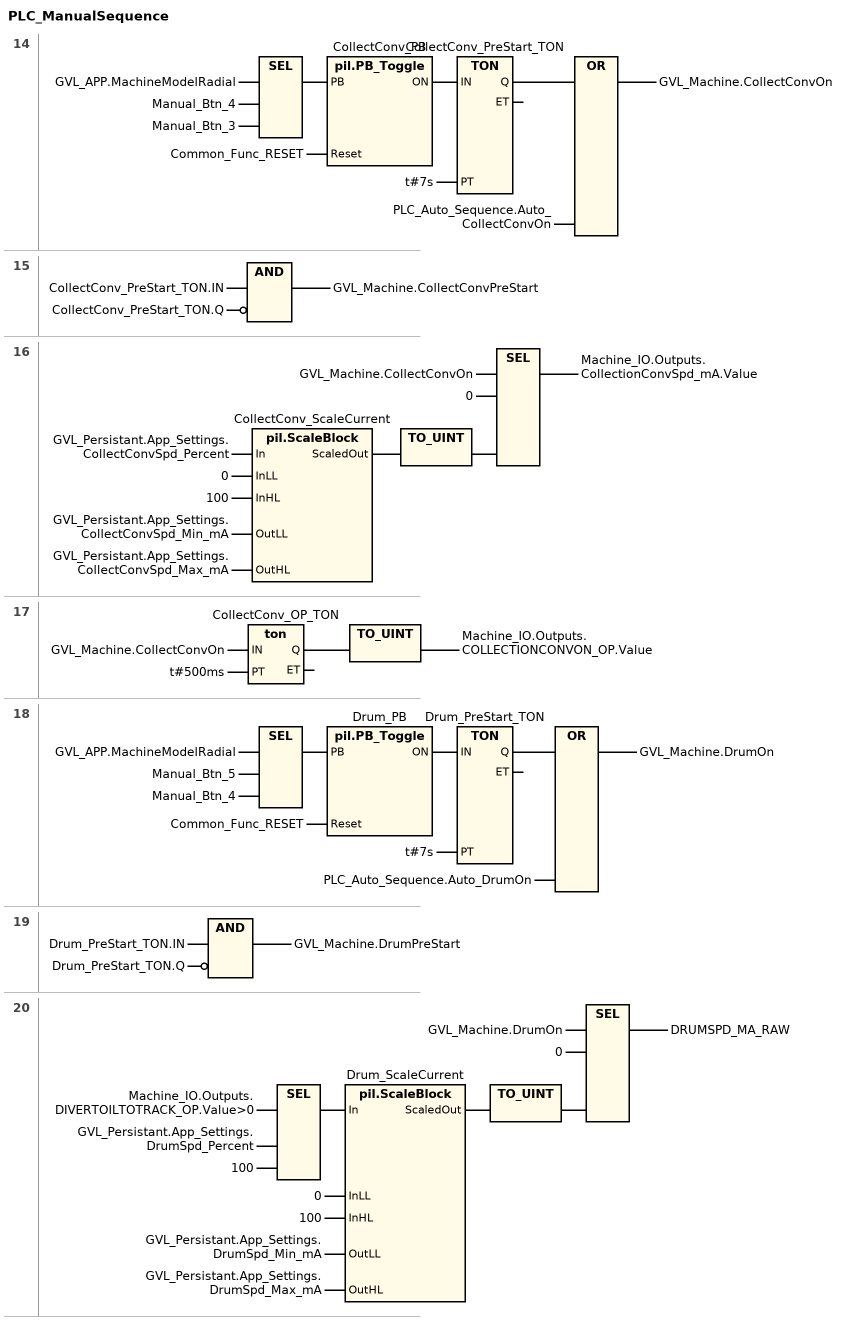
// NETWORK 14
CollectConv_PB(PB := SEL(GVL_APP.MachineModelRadial, Manual_Btn_4, Manual_Btn_3), Reset := Common_Func_RESET); // pil.PB_Toggle
CollectConv_PreStart_TON(IN := CollectConv_PB.ON, PT := t#7s); // TON
GVL_Machine.CollectConvOn := CollectConv_PreStart_TON.Q OR PLC_Auto_Sequence.Auto_CollectConvOn;

// NETWORK 15
GVL_Machine.CollectConvPreStart := CollectConv_PreStart_TON.IN AND NOT CollectConv_PreStart_TON.Q;

// NETWORK 16
CollectConv_ScaleCurrent(
    In := GVL_Persistant.App_Settings.CollectConvSpd_Percent,
    InLL := 0,
    InHL := 100,
    OutLL := GVL_Persistant.App_Settings.CollectConvSpd_Min_mA,
    OutHL := GVL_Persistant.App_Settings.CollectConvSpd_Max_mA); // pil.ScaleBlock
Machine_IO.Outputs.CollectionConvSpd_mA.Value := SEL(GVL_Machine.CollectConvOn, 0, TO_UINT(CollectConv_ScaleCurrent.ScaledOut));

// NETWORK 17
CollectConv_OP_TON(IN := GVL_Machine.CollectConvOn, PT := t#500ms); // ton
Machine_IO.Outputs.COLLECTIONCONVON_OP.Value := TO_UINT(CollectConv_OP_TON.Q);

// NETWORK 18
Drum_PB(PB := SEL(GVL_APP.MachineModelRadial, Manual_Btn_5, Manual_Btn_4), Reset := Common_Func_RESET); // pil.PB_Toggle
Drum_PreStart_TON(IN := Drum_PB.ON, PT := t#7s); // TON
GVL_Machine.DrumOn := Drum_PreStart_TON.Q OR PLC_Auto_Sequence.Auto_DrumOn;

// NETWORK 19
GVL_Machine.DrumPreStart := Drum_PreStart_TON.IN AND NOT Drum_PreStart_TON.Q;

// NETWORK 20
Drum_ScaleCurrent(
    In := SEL(Machine_IO.Outputs.DIVERTOILTOTRACK_OP.Value>0, GVL_Persistant.App_Settings.DrumSpd_Percent, 100),
    InLL := 0,
    InHL := 100,
    OutLL := GVL_Persistant.App_Settings.DrumSpd_Min_mA,
    OutHL := GVL_Persistant.App_Settings.DrumSpd_Max_mA); // pil.ScaleBlock
DRUMSPD_MA_RAW := SEL(GVL_Machine.DrumOn, 0, TO_UINT(Drum_ScaleCurrent.ScaledOut));

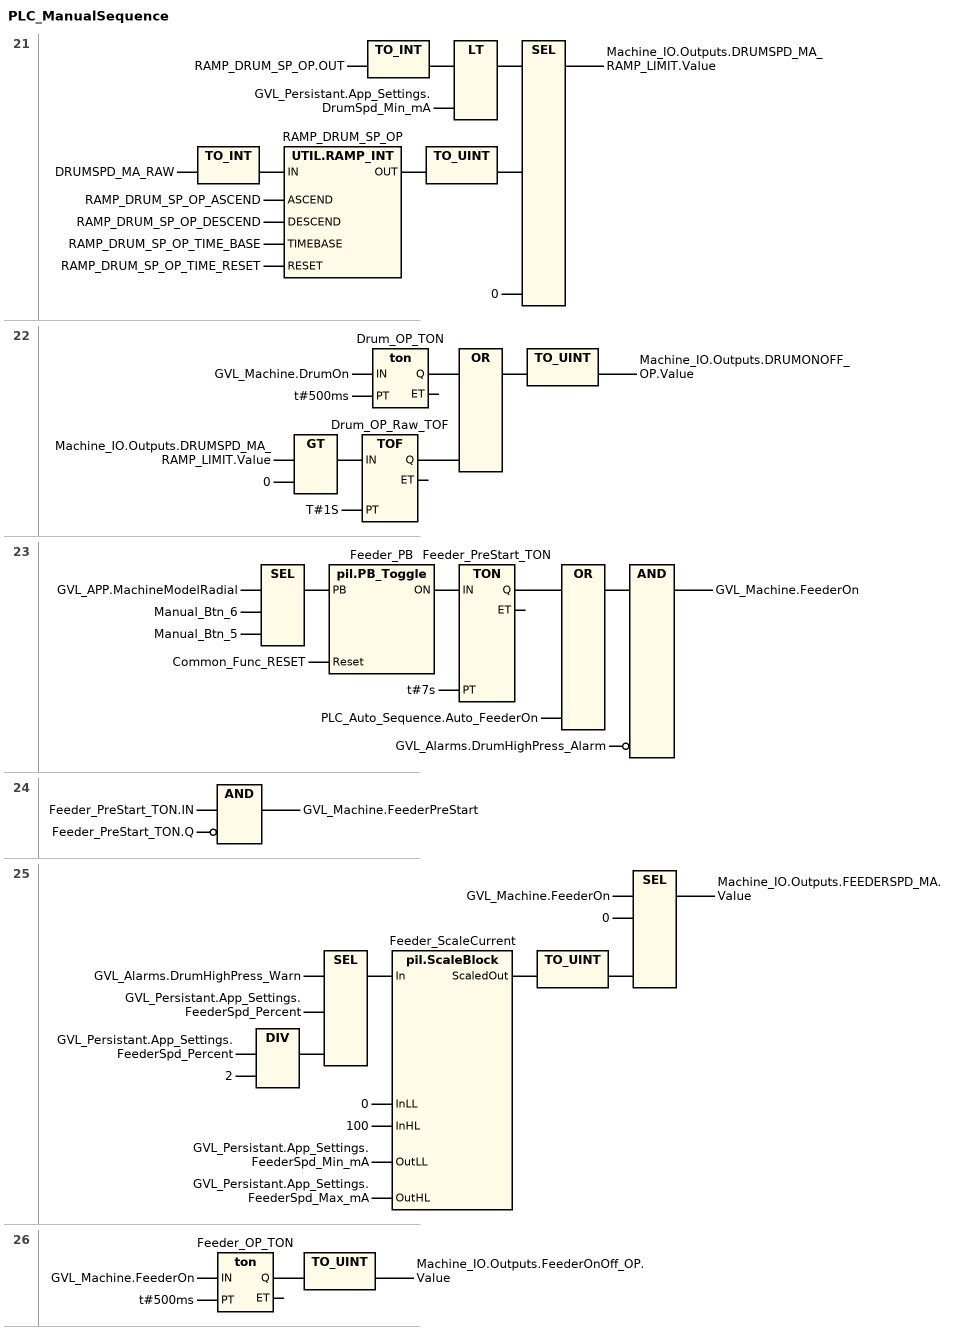
// NETWORK 21
_w1 := TO_INT(RAMP_DRUM_SP_OP.OUT) < GVL_Persistant.App_Settings.DrumSpd_Min_mA;
RAMP_DRUM_SP_OP(
    IN := TO_INT(DRUMSPD_MA_RAW),
    ASCEND := RAMP_DRUM_SP_OP_ASCEND,
    DESCEND := RAMP_DRUM_SP_OP_DESCEND,
    TIMEBASE := RAMP_DRUM_SP_OP_TIME_BASE,
    RESET := RAMP_DRUM_SP_OP_TIME_RESET); // UTIL.RAMP_INT
Machine_IO.Outputs.DRUMSPD_MA_RAMP_LIMIT.Value := SEL(_w1, TO_UINT(RAMP_DRUM_SP_OP.OUT), 0);

// NETWORK 22
Drum_OP_TON(IN := GVL_Machine.DrumOn, PT := t#500ms); // ton
Drum_OP_Raw_TOF(IN := Machine_IO.Outputs.DRUMSPD_MA_RAMP_LIMIT.Value > 0, PT := T#1S); // TOF
Machine_IO.Outputs.DRUMONOFF_OP.Value := TO_UINT(Drum_OP_TON.Q OR Drum_OP_Raw_TOF.Q);

// NETWORK 23
Feeder_PB(PB := SEL(GVL_APP.MachineModelRadial, Manual_Btn_6, Manual_Btn_5), Reset := Common_Func_RESET); // pil.PB_Toggle
Feeder_PreStart_TON(IN := Feeder_PB.ON, PT := t#7s); // TON
GVL_Machine.FeederOn := (Feeder_PreStart_TON.Q OR PLC_Auto_Sequence.Auto_FeederOn) AND NOT GVL_Alarms.DrumHighPress_Alarm;

// NETWORK 24
GVL_Machine.FeederPreStart := Feeder_PreStart_TON.IN AND NOT Feeder_PreStart_TON.Q;

// NETWORK 25
Feeder_ScaleCurrent(
    In := SEL(GVL_Alarms.DrumHighPress_Warn, GVL_Persistant.App_Settings.FeederSpd_Percent, GVL_Persistant.App_Settings.FeederSpd_Percent / 2),
    InLL := 0,
    InHL := 100,
    OutLL := GVL_Persistant.App_Settings.FeederSpd_Min_mA,
    OutHL := GVL_Persistant.App_Settings.FeederSpd_Max_mA); // pil.ScaleBlock
Machine_IO.Outputs.FEEDERSPD_MA.Value := SEL(GVL_Machine.FeederOn, 0, TO_UINT(Feeder_ScaleCurrent.ScaledOut));

// NETWORK 26
Feeder_OP_TON(IN := GVL_Machine.FeederOn, PT := t#500ms); // ton
Machine_IO.Outputs.FeederOnOff_OP.Value := TO_UINT(Feeder_OP_TON.Q);

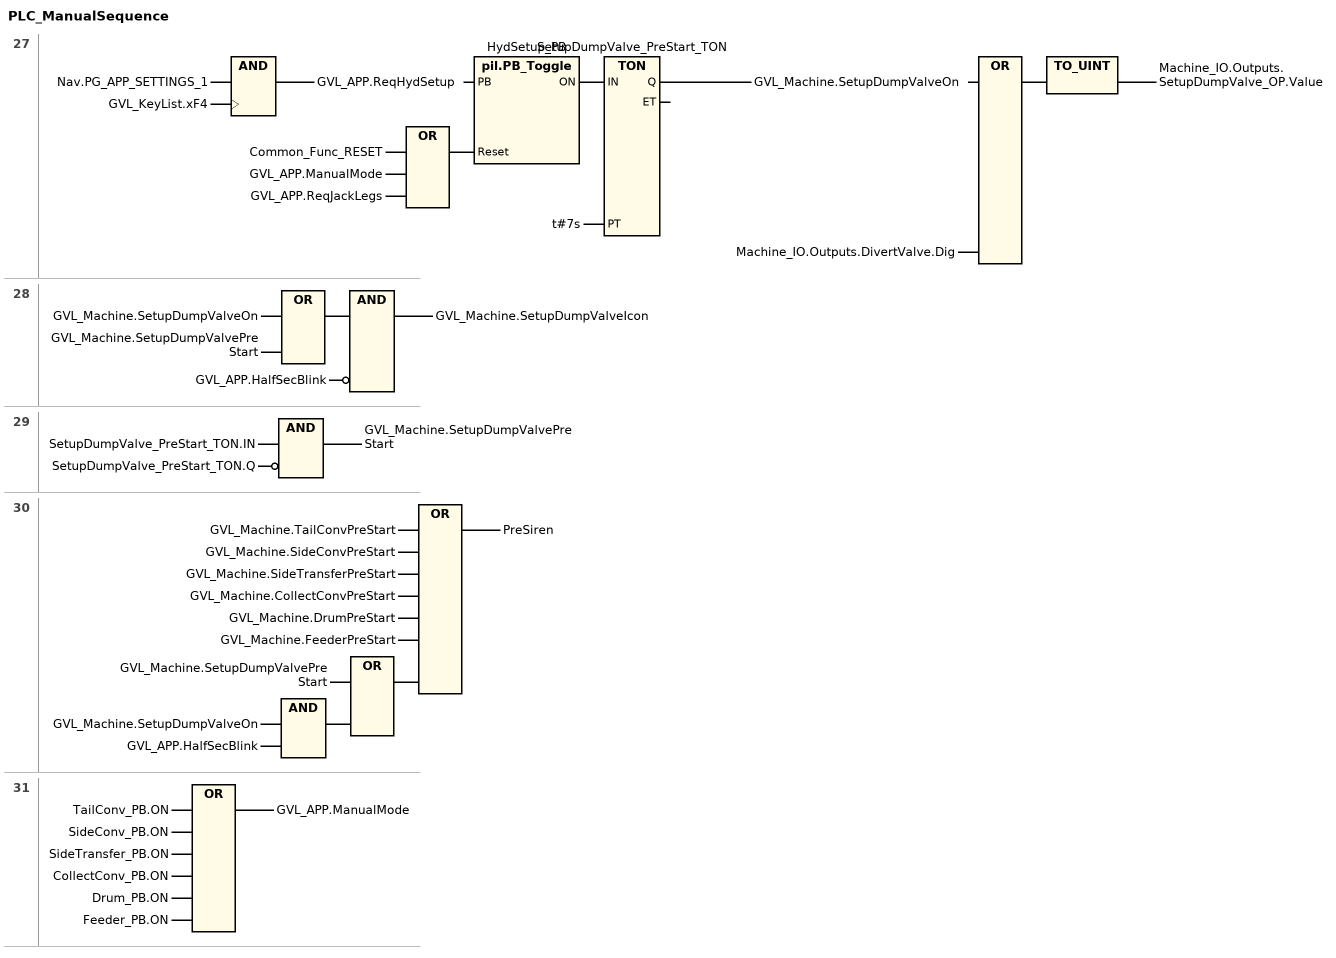
// NETWORK 27
_rt1(CLK := GVL_KeyList.xF4);
_w2 := Nav.PG_APP_SETTINGS_1 AND _rt1.Q;
GVL_APP.ReqHydSetup := _w2;
HydSetup_PB(PB := _w2, Reset := Common_Func_RESET OR GVL_APP.ManualMode OR GVL_APP.ReqJackLegs); // pil.PB_Toggle
SetupDumpValve_PreStart_TON(IN := HydSetup_PB.ON, PT := t#7s); // TON
GVL_Machine.SetupDumpValveOn := SetupDumpValve_PreStart_TON.Q;
Machine_IO.Outputs.SetupDumpValve_OP.Value := TO_UINT(SetupDumpValve_PreStart_TON.Q OR Machine_IO.Outputs.DivertValve.Dig);

// NETWORK 28
GVL_Machine.SetupDumpValveIcon := (GVL_Machine.SetupDumpValveOn OR GVL_Machine.SetupDumpValvePreStart) AND NOT GVL_APP.HalfSecBlink;

// NETWORK 29
GVL_Machine.SetupDumpValvePreStart := SetupDumpValve_PreStart_TON.IN AND NOT SetupDumpValve_PreStart_TON.Q;

// NETWORK 30
PreSiren := GVL_Machine.TailConvPreStart OR GVL_Machine.SideConvPreStart OR GVL_Machine.SideTransferPreStart OR GVL_Machine.CollectConvPreStart OR GVL_Machine.DrumPreStart OR GVL_Machine.FeederPreStart OR (GVL_Machine.SetupDumpValvePreStart OR GVL_Machine.SetupDumpValveOn AND GVL_APP.HalfSecBlink);

// NETWORK 31
GVL_APP.ManualMode := TailConv_PB.ON OR SideConv_PB.ON OR SideTransfer_PB.ON OR CollectConv_PB.ON OR Drum_PB.ON OR Feeder_PB.ON;

END_PROGRAM

// Device/Application/App_PLC/Control/PLC_Auto_Sequence
PROGRAM PLC_Auto_Sequence
VAR
	AutoStopMode_Toggle: pil.PB_Toggle;
	AutoSequence_Toggle: pil.PB_Toggle;

	PrestartTon: TON;
	PreSiren: BOOL;
	AutoStarting: BOOL;
	
	TailConv_PB: pil.PB_Toggle;
	WaitToStopTailConv_TON: TON;
	Auto_TailConvOn: BOOL;
	
	WaitToStartSideConv_TON: TON;
	WaitToStopSideConv_TON: TON;	
	SideConv_PB: pil.PB_Toggle;
	Auto_SideConvOn: BOOL;
	
	WaitToStartSideTransfer_TON: TON;
	WaitToStopSideTransfer_TON: TON;
	SideTransfer_PB: pil.PB_Toggle;
	Auto_SideTransferOn: BOOL;
	
	WaitToStartCollectConv_TON: TON;
	WaitToStopCollectConv_TON: TON;
	CollectConv_PB: pil.PB_Toggle;
	Auto_CollectConvOn: BOOL;
	
	WaitToStartDrum_TON: TON;
	WaitToStopDrum_TON: TON;
	Drum_PB: pil.PB_Toggle;
	Auto_DrumOn: BOOL;
	
	WaitToFeeder_TON: TON;
	WaitToStopFeeder_TON: TON;	
	Feeder_PB: pil.PB_Toggle;
	Auto_FeederOn: BOOL;
	StartUpComplete: BOOL;
	
	F_TRIG_0: f_trig;
	F_TRIG_1: f_trig;
	
	Common_Func_RESET: BOOL;
END_VAR
VAR RETAIN
END_VAR

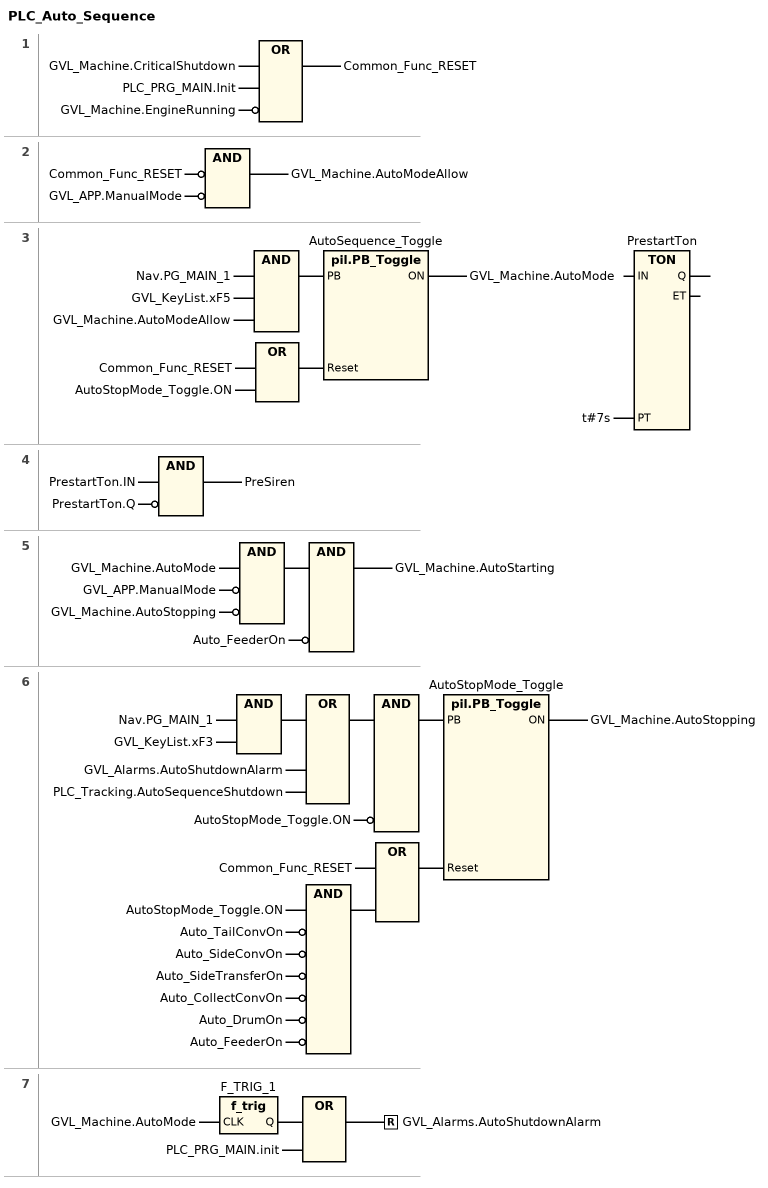
// NETWORK 1
Common_Func_RESET := GVL_Machine.CriticalShutdown OR PLC_PRG_MAIN.Init OR NOT GVL_Machine.EngineRunning;

// NETWORK 2
GVL_Machine.AutoModeAllow := NOT Common_Func_RESET AND NOT GVL_APP.ManualMode;

// NETWORK 3
AutoSequence_Toggle(PB := Nav.PG_MAIN_1 AND GVL_KeyList.xF5 AND GVL_Machine.AutoModeAllow, Reset := Common_Func_RESET OR AutoStopMode_Toggle.ON); // pil.PB_Toggle
GVL_Machine.AutoMode := AutoSequence_Toggle.ON;
PrestartTon(IN := AutoSequence_Toggle.ON, PT := t#7s); // TON

// NETWORK 4
PreSiren := PrestartTon.IN AND NOT PrestartTon.Q;

// NETWORK 5
GVL_Machine.AutoStarting := (GVL_Machine.AutoMode AND NOT GVL_APP.ManualMode AND NOT GVL_Machine.AutoStopping) AND NOT Auto_FeederOn;

// NETWORK 6
AutoStopMode_Toggle(PB := (Nav.PG_MAIN_1 AND GVL_KeyList.xF3 OR GVL_Alarms.AutoShutdownAlarm OR PLC_Tracking.AutoSequenceShutdown) AND NOT AutoStopMode_Toggle.ON, Reset := Common_Func_RESET OR AutoStopMode_Toggle.ON AND NOT Auto_TailConvOn AND NOT Auto_SideConvOn AND NOT Auto_SideTransferOn AND NOT Auto_CollectConvOn AND NOT Auto_DrumOn AND NOT Auto_FeederOn); // pil.PB_Toggle
GVL_Machine.AutoStopping := AutoStopMode_Toggle.ON;

// NETWORK 7
F_TRIG_1(CLK := GVL_Machine.AutoMode); // f_trig
GVL_Alarms.AutoShutdownAlarm R= F_TRIG_1.Q OR PLC_PRG_MAIN.init;

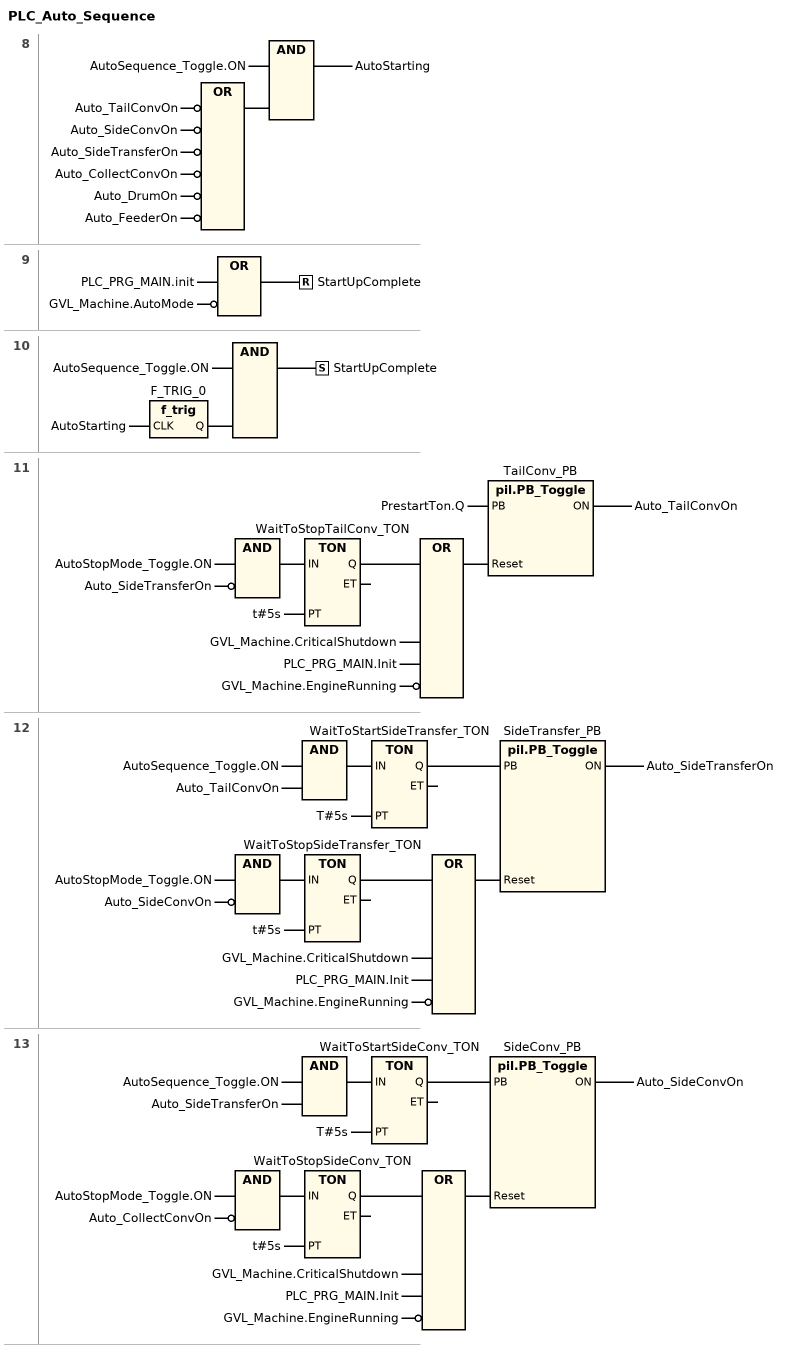
// NETWORK 8
AutoStarting := AutoSequence_Toggle.ON AND (NOT Auto_TailConvOn OR NOT Auto_SideConvOn OR NOT Auto_SideTransferOn OR NOT Auto_CollectConvOn OR NOT Auto_DrumOn OR NOT Auto_FeederOn);

// NETWORK 9
StartUpComplete R= PLC_PRG_MAIN.init OR NOT GVL_Machine.AutoMode;

// NETWORK 10
F_TRIG_0(CLK := AutoStarting); // f_trig
StartUpComplete S= AutoSequence_Toggle.ON AND F_TRIG_0.Q;

// NETWORK 11
WaitToStopTailConv_TON(IN := AutoStopMode_Toggle.ON AND NOT Auto_SideTransferOn, PT := t#5s); // TON
TailConv_PB(PB := PrestartTon.Q, Reset := WaitToStopTailConv_TON.Q OR GVL_Machine.CriticalShutdown OR PLC_PRG_MAIN.Init OR NOT GVL_Machine.EngineRunning); // pil.PB_Toggle
Auto_TailConvOn := TailConv_PB.ON;

// NETWORK 12
WaitToStartSideTransfer_TON(IN := AutoSequence_Toggle.ON AND Auto_TailConvOn, PT := T#5s); // TON
WaitToStopSideTransfer_TON(IN := AutoStopMode_Toggle.ON AND NOT Auto_SideConvOn, PT := t#5s); // TON
SideTransfer_PB(PB := WaitToStartSideTransfer_TON.Q, Reset := WaitToStopSideTransfer_TON.Q OR GVL_Machine.CriticalShutdown OR PLC_PRG_MAIN.Init OR NOT GVL_Machine.EngineRunning); // pil.PB_Toggle
Auto_SideTransferOn := SideTransfer_PB.ON;

// NETWORK 13
WaitToStartSideConv_TON(IN := AutoSequence_Toggle.ON AND Auto_SideTransferOn, PT := T#5s); // TON
WaitToStopSideConv_TON(IN := AutoStopMode_Toggle.ON AND NOT Auto_CollectConvOn, PT := t#5s); // TON
SideConv_PB(PB := WaitToStartSideConv_TON.Q, Reset := WaitToStopSideConv_TON.Q OR GVL_Machine.CriticalShutdown OR PLC_PRG_MAIN.Init OR NOT GVL_Machine.EngineRunning); // pil.PB_Toggle
Auto_SideConvOn := SideConv_PB.ON;

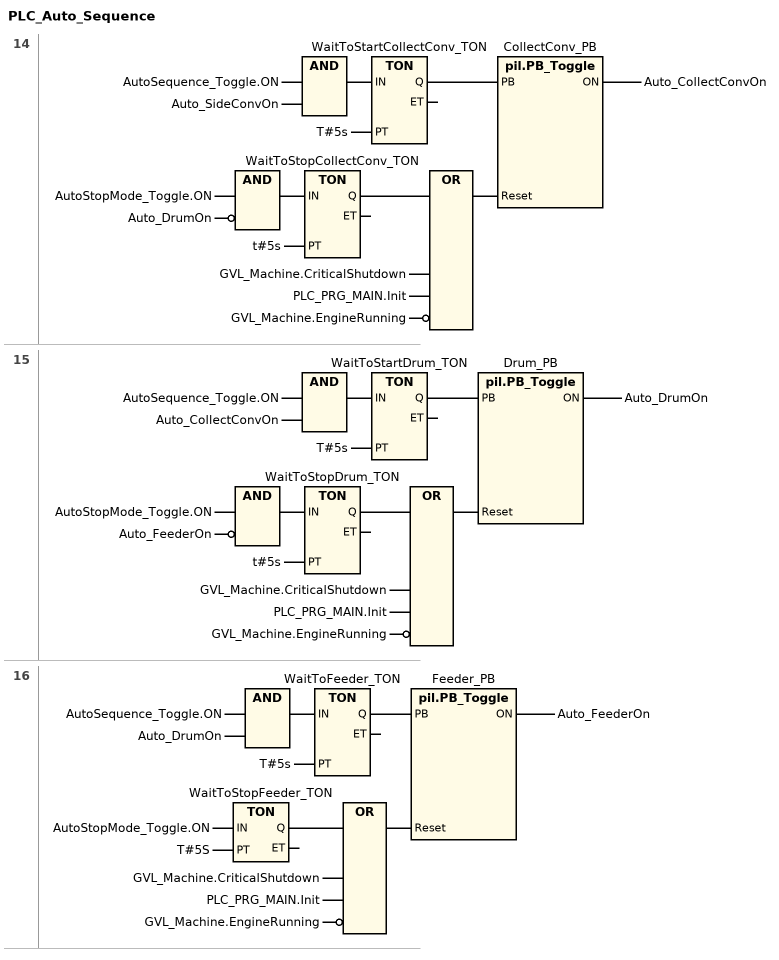
// NETWORK 14
WaitToStartCollectConv_TON(IN := AutoSequence_Toggle.ON AND Auto_SideConvOn, PT := T#5s); // TON
WaitToStopCollectConv_TON(IN := AutoStopMode_Toggle.ON AND NOT Auto_DrumOn, PT := t#5s); // TON
CollectConv_PB(PB := WaitToStartCollectConv_TON.Q, Reset := WaitToStopCollectConv_TON.Q OR GVL_Machine.CriticalShutdown OR PLC_PRG_MAIN.Init OR NOT GVL_Machine.EngineRunning); // pil.PB_Toggle
Auto_CollectConvOn := CollectConv_PB.ON;

// NETWORK 15
WaitToStartDrum_TON(IN := AutoSequence_Toggle.ON AND Auto_CollectConvOn, PT := T#5s); // TON
WaitToStopDrum_TON(IN := AutoStopMode_Toggle.ON AND NOT Auto_FeederOn, PT := t#5s); // TON
Drum_PB(PB := WaitToStartDrum_TON.Q, Reset := WaitToStopDrum_TON.Q OR GVL_Machine.CriticalShutdown OR PLC_PRG_MAIN.Init OR NOT GVL_Machine.EngineRunning); // pil.PB_Toggle
Auto_DrumOn := Drum_PB.ON;

// NETWORK 16
WaitToFeeder_TON(IN := AutoSequence_Toggle.ON AND Auto_DrumOn, PT := T#5s); // TON
WaitToStopFeeder_TON(IN := AutoStopMode_Toggle.ON, PT := T#5S); // TON
Feeder_PB(PB := WaitToFeeder_TON.Q, Reset := WaitToStopFeeder_TON.Q OR GVL_Machine.CriticalShutdown OR PLC_PRG_MAIN.Init OR NOT GVL_Machine.EngineRunning); // pil.PB_Toggle
Auto_FeederOn := Feeder_PB.ON;

END_PROGRAM

// Device/Application/App_PLC/Control/PLC_Tracking
PROGRAM PLC_Tracking
VAR
	TrackingEnabled_Toggle: PIL.PB_Toggle;
	Track_PreSiren_TON: TON;
	Prestart: BOOL;

	AutoSequenceShutdown: BOOL;
	EngineRampDownSet: BOOL;
	EngineSetTrackingRpm: BOOL;
	R_TRIG_0: r_TRig;
	WaitTon_1: TON;
	PreSiren_Cancel: BOOL;
	TRACK_PRESIREN_FLASH: DUTY_CYCLE;
	TrackingModeAllow_Toggle: PIL.PB_Toggle;
	TRACKING_COMMON_STOP: BOOL;
END_VAR

VAR_OUTPUT
	Siren: BOOL;
END_VAR
VAR // added by the converter: edge detectors and wires of the graphical bodies
    _rt1 : R_TRIG;
END_VAR

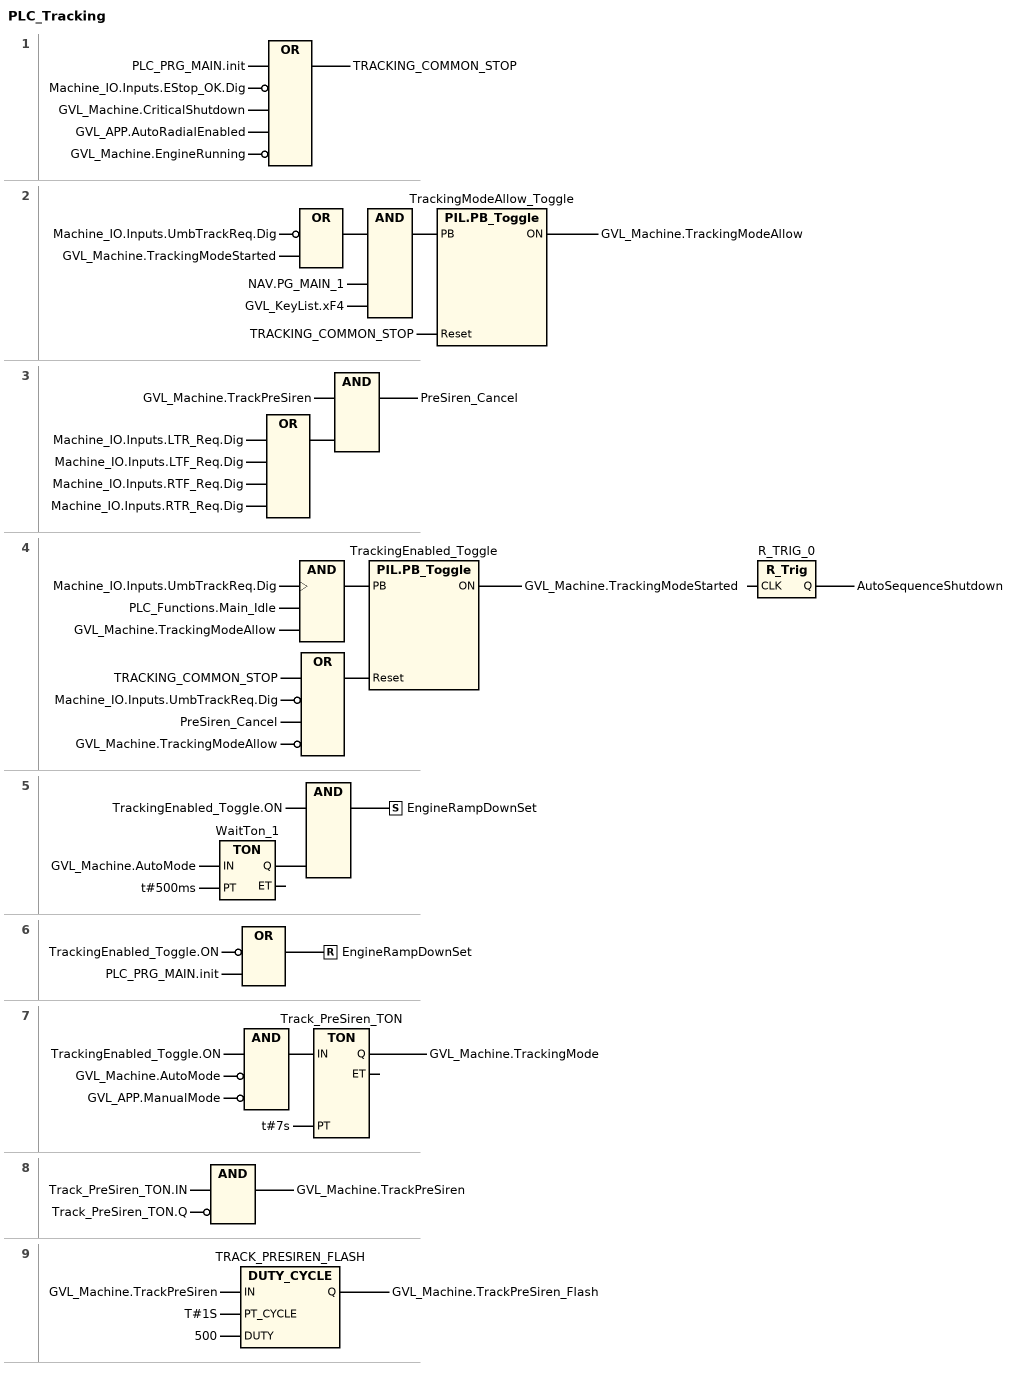
// NETWORK 1
TRACKING_COMMON_STOP := PLC_PRG_MAIN.init OR NOT Machine_IO.Inputs.EStop_OK.Dig OR GVL_Machine.CriticalShutdown OR GVL_APP.AutoRadialEnabled OR NOT GVL_Machine.EngineRunning;

// NETWORK 2
TrackingModeAllow_Toggle(PB := (NOT Machine_IO.Inputs.UmbTrackReq.Dig OR GVL_Machine.TrackingModeStarted) AND NAV.PG_MAIN_1 AND GVL_KeyList.xF4, Reset := TRACKING_COMMON_STOP); // PIL.PB_Toggle
GVL_Machine.TrackingModeAllow := TrackingModeAllow_Toggle.ON;

// NETWORK 3
PreSiren_Cancel := GVL_Machine.TrackPreSiren AND (Machine_IO.Inputs.LTR_Req.Dig OR Machine_IO.Inputs.LTF_Req.Dig OR Machine_IO.Inputs.RTF_Req.Dig OR Machine_IO.Inputs.RTR_Req.Dig);

// NETWORK 4
_rt1(CLK := Machine_IO.Inputs.UmbTrackReq.Dig);
TrackingEnabled_Toggle(PB := _rt1.Q AND PLC_Functions.Main_Idle AND GVL_Machine.TrackingModeAllow, Reset := TRACKING_COMMON_STOP OR NOT Machine_IO.Inputs.UmbTrackReq.Dig OR PreSiren_Cancel OR NOT GVL_Machine.TrackingModeAllow); // PIL.PB_Toggle
GVL_Machine.TrackingModeStarted := TrackingEnabled_Toggle.ON;
R_TRIG_0(CLK := TrackingEnabled_Toggle.ON); // R_Trig
AutoSequenceShutdown := R_TRIG_0.Q;

// NETWORK 5
WaitTon_1(IN := GVL_Machine.AutoMode, PT := t#500ms); // TON
EngineRampDownSet S= TrackingEnabled_Toggle.ON AND WaitTon_1.Q;

// NETWORK 6
EngineRampDownSet R= NOT TrackingEnabled_Toggle.ON OR PLC_PRG_MAIN.init;

// NETWORK 7
Track_PreSiren_TON(IN := TrackingEnabled_Toggle.ON AND NOT GVL_Machine.AutoMode AND NOT GVL_APP.ManualMode, PT := t#7s); // TON
GVL_Machine.TrackingMode := Track_PreSiren_TON.Q;

// NETWORK 8
GVL_Machine.TrackPreSiren := Track_PreSiren_TON.IN AND NOT Track_PreSiren_TON.Q;

// NETWORK 9
TRACK_PRESIREN_FLASH(IN := GVL_Machine.TrackPreSiren, PT_CYCLE := T#1S, DUTY := 500); // DUTY_CYCLE
GVL_Machine.TrackPreSiren_Flash := TRACK_PRESIREN_FLASH.Q;

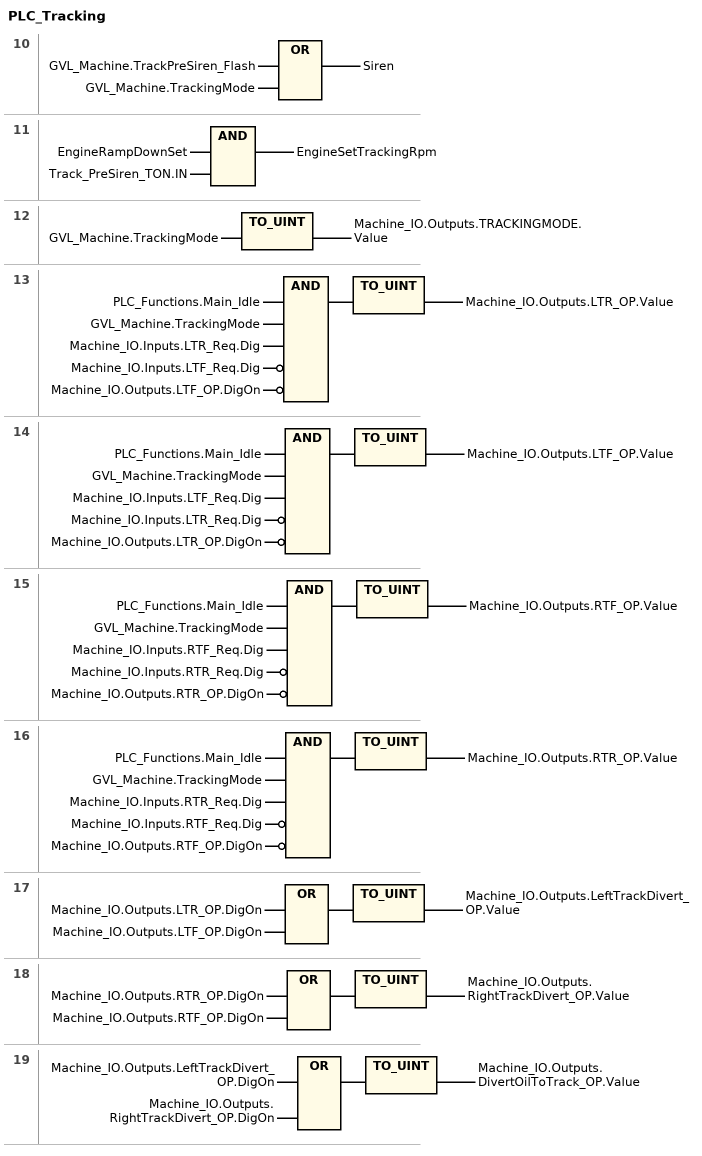
// NETWORK 10
Siren := GVL_Machine.TrackPreSiren_Flash OR GVL_Machine.TrackingMode;

// NETWORK 11
EngineSetTrackingRpm := EngineRampDownSet AND Track_PreSiren_TON.IN;

// NETWORK 12
Machine_IO.Outputs.TRACKINGMODE.Value := TO_UINT(GVL_Machine.TrackingMode);

// NETWORK 13
Machine_IO.Outputs.LTR_OP.Value := TO_UINT(PLC_Functions.Main_Idle AND GVL_Machine.TrackingMode AND Machine_IO.Inputs.LTR_Req.Dig AND NOT Machine_IO.Inputs.LTF_Req.Dig AND NOT Machine_IO.Outputs.LTF_OP.DigOn);

// NETWORK 14
Machine_IO.Outputs.LTF_OP.Value := TO_UINT(PLC_Functions.Main_Idle AND GVL_Machine.TrackingMode AND Machine_IO.Inputs.LTF_Req.Dig AND NOT Machine_IO.Inputs.LTR_Req.Dig AND NOT Machine_IO.Outputs.LTR_OP.DigOn);

// NETWORK 15
Machine_IO.Outputs.RTF_OP.Value := TO_UINT(PLC_Functions.Main_Idle AND GVL_Machine.TrackingMode AND Machine_IO.Inputs.RTF_Req.Dig AND NOT Machine_IO.Inputs.RTR_Req.Dig AND NOT Machine_IO.Outputs.RTR_OP.DigOn);

// NETWORK 16
Machine_IO.Outputs.RTR_OP.Value := TO_UINT(PLC_Functions.Main_Idle AND GVL_Machine.TrackingMode AND Machine_IO.Inputs.RTR_Req.Dig AND NOT Machine_IO.Inputs.RTF_Req.Dig AND NOT Machine_IO.Outputs.RTF_OP.DigOn);

// NETWORK 17
Machine_IO.Outputs.LeftTrackDivert_OP.Value := TO_UINT(Machine_IO.Outputs.LTR_OP.DigOn OR Machine_IO.Outputs.LTF_OP.DigOn);

// NETWORK 18
Machine_IO.Outputs.RightTrackDivert_OP.Value := TO_UINT(Machine_IO.Outputs.RTR_OP.DigOn OR Machine_IO.Outputs.RTF_OP.DigOn);

// NETWORK 19
Machine_IO.Outputs.DivertOilToTrack_OP.Value := TO_UINT(Machine_IO.Outputs.LeftTrackDivert_OP.DigOn OR Machine_IO.Outputs.RightTrackDivert_OP.DigOn);

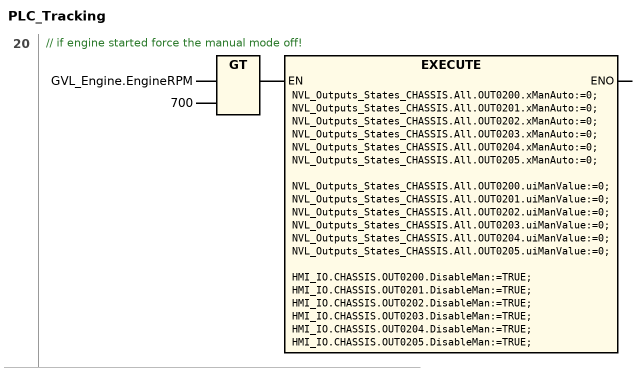
// NETWORK 20
// // if engine started force the manual mode off!
IF GVL_Engine.EngineRPM > 700 THEN
    NVL_Outputs_States_CHASSIS.All.OUT0200.xManAuto:=0;
    NVL_Outputs_States_CHASSIS.All.OUT0201.xManAuto:=0;
    NVL_Outputs_States_CHASSIS.All.OUT0202.xManAuto:=0;
    NVL_Outputs_States_CHASSIS.All.OUT0203.xManAuto:=0;
    NVL_Outputs_States_CHASSIS.All.OUT0204.xManAuto:=0;
    NVL_Outputs_States_CHASSIS.All.OUT0205.xManAuto:=0;
    
    NVL_Outputs_States_CHASSIS.All.OUT0200.uiManValue:=0;
    NVL_Outputs_States_CHASSIS.All.OUT0201.uiManValue:=0;
    NVL_Outputs_States_CHASSIS.All.OUT0202.uiManValue:=0;
    NVL_Outputs_States_CHASSIS.All.OUT0203.uiManValue:=0;
    NVL_Outputs_States_CHASSIS.All.OUT0204.uiManValue:=0;
    NVL_Outputs_States_CHASSIS.All.OUT0205.uiManValue:=0;
    
    HMI_IO.CHASSIS.OUT0200.DisableMan:=TRUE;
    HMI_IO.CHASSIS.OUT0201.DisableMan:=TRUE;
    HMI_IO.CHASSIS.OUT0202.DisableMan:=TRUE;
    HMI_IO.CHASSIS.OUT0203.DisableMan:=TRUE;
    HMI_IO.CHASSIS.OUT0204.DisableMan:=TRUE;
    HMI_IO.CHASSIS.OUT0205.DisableMan:=TRUE;
END_IF

END_PROGRAM

// Device/Application/App_PLC/Control/PLC_Functions
PROGRAM PLC_Functions
VAR
	Main_Idle_TON: TON;
	Engine_Idle_TON: TON;
END_VAR

VAR_OUTPUT
	Main_Idle:BOOL;
	Engine_Idle:BOOL;
END_VAR

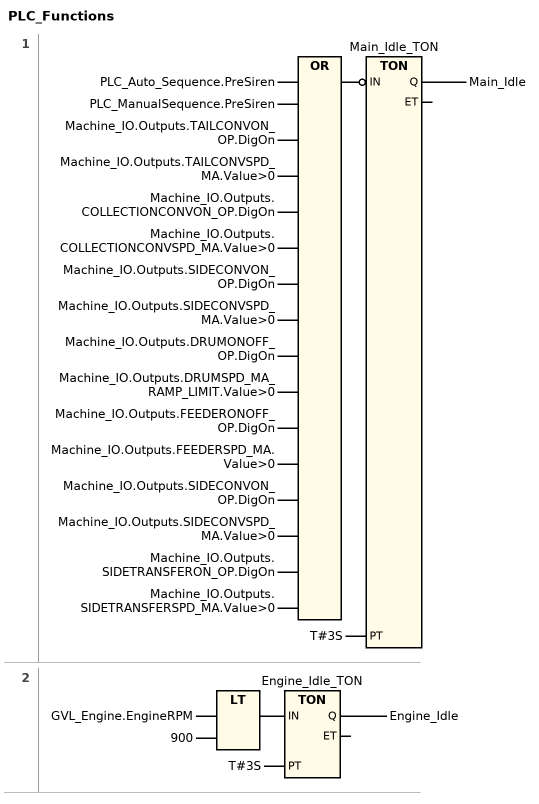
// NETWORK 1
Main_Idle_TON(IN := NOT (PLC_Auto_Sequence.PreSiren OR PLC_ManualSequence.PreSiren OR Machine_IO.Outputs.TAILCONVON_OP.DigOn OR (Machine_IO.Outputs.TAILCONVSPD_MA.Value>0) OR Machine_IO.Outputs.COLLECTIONCONVON_OP.DigOn OR (Machine_IO.Outputs.COLLECTIONCONVSPD_MA.Value>0) OR Machine_IO.Outputs.SIDECONVON_OP.DigOn OR (Machine_IO.Outputs.SIDECONVSPD_MA.Value>0) OR Machine_IO.Outputs.DRUMONOFF_OP.DigOn OR (Machine_IO.Outputs.DRUMSPD_MA_RAMP_LIMIT.Value>0) OR Machine_IO.Outputs.FEEDERONOFF_OP.DigOn OR (Machine_IO.Outputs.FEEDERSPD_MA.Value>0) OR Machine_IO.Outputs.SIDECONVON_OP.DigOn OR (Machine_IO.Outputs.SIDECONVSPD_MA.Value>0) OR Machine_IO.Outputs.SIDETRANSFERON_OP.DigOn OR (Machine_IO.Outputs.SIDETRANSFERSPD_MA.Value>0)), PT := T#3S); // TON
Main_Idle := Main_Idle_TON.Q;

// NETWORK 2
Engine_Idle_TON(IN := GVL_Engine.EngineRPM < 900, PT := T#3S); // TON
Engine_Idle := Engine_Idle_TON.Q;

END_PROGRAM

// Device/Application/App_PLC/Control/PLC_RadialMode
PROGRAM PLC_RadialMode
VAR
	EnableRadialBtn: pil.PB_Toggle;
	PreStart_TON: ton;
	Timed_Radial: pil.PB_Toggle;
	Radial_TimeOut_Ton: ton;
	Radial_Time_Delay: ton;
	Auto_PreSiren: BOOL;
	Radial_LeftToggle: pil.PB_Toggle;
	RadialRightOn: tof;
	AutoRight_OP: BOOL;
	RadialLeftOn: tof;
	AutoLeft_OP: BOOL;
	Man_Move_PreStart_TON: ton;
	ManualRadialReq: BOOL;
	Manual_Move_PreSiren: BOOL;
	Siren: BOOL;
	INIT_LOCAL: BOOL := TRUE;
	Radial_TimeOut_Secs: DWORD;
	Radial_TimeDelay_Secs: DWORD;
	MANUAL_FORCE_RADIAL: BOOL;
	Left_Radial_Switch_TON: TON;
	Right_Radial_Switch_TON: TON;
	Left_Limit_Swt_Active: BOOL;
	Right_Limit_Swt_Active: BOOL;
	Man_Left_Move: BOOL;
	Man_Right_Move: BOOL;
END_VAR

VAR_OUTPUT
	RadialLeft_OP: BOOL;
	RadialRight_OP: BOOL;
	STATUS_STRING: STRING;
END_VAR
VAR // added by the converter: edge detectors and wires of the graphical bodies
    _rt1, _rt2, _rt3, _rt4, _rt5 : R_TRIG;
    _ft1 : F_TRIG;
    _w1, _w2, _w3 : BOOL;
END_VAR

